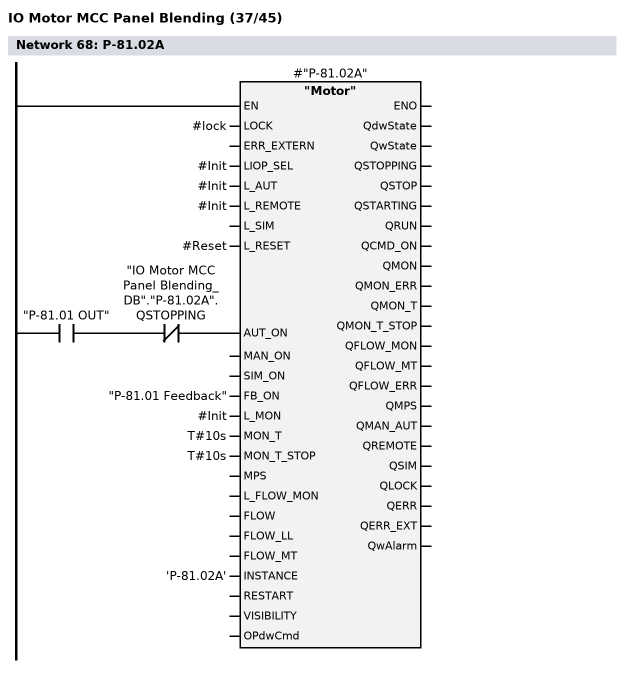
   RUNG wire#powerrail
      #"P-81.02A"(AUT_ON := wire#w1, LOCK := #lock, ERR_EXTERN :=, LIOP_SEL := #Init, L_AUT := #Init, L_REMOTE := #Init, L_SIM :=, L_RESET := #Reset, MAN_ON :=, SIM_ON :=, FB_ON := "P-81.01 Feedback", L_MON := #Init, MON_T := T#10s, MON_T_STOP := T#10s, MPS :=, L_FLOW_MON :=, FLOW :=, FLOW_LL :=, FLOW_MT :=, INSTANCE := 'P-81.02A', RESTART :=, VISIBILITY :=, OPdwCmd :=, QdwState =>, QwState =>, QSTOPPING =>, QSTOP =>, QSTARTING =>, QRUN =>, QCMD_ON =>, QMON =>, QMON_ERR =>, QMON_T =>, QMON_T_STOP =>, QFLOW_MON =>, QFLOW_MT =>, QFLOW_ERR =>, QMPS =>, QMAN_AUT =>, QREMOTE =>, QSIM =>, QLOCK =>, QERR =>, QERR_EXT =>, QwAlarm =>)
   END_RUNG
   RUNG wire#powerrail
      Contact( "P-81.01 OUT" )
      I_Contact( "IO Motor MCC Panel Blending_DB"."P-81.02A".QSTOPPING )
   END_RUNG wire#w1
   // the same network as SCL:
   #"P-81.02A"(LOCK := #lock,   // "Motor"
               LIOP_SEL := #Init,
               L_AUT := #Init,
               L_REMOTE := #Init,
               L_RESET := #Reset,
               AUT_ON := "P-81.01 OUT" AND NOT "IO Motor MCC Panel Blending_DB"."P-81.02A".QSTOPPING,
               FB_ON := "P-81.01 Feedback",
               L_MON := #Init,
               MON_T := T#10s,
               MON_T_STOP := T#10s,
               INSTANCE := 'P-81.02A');
END_REGION

REGION Network 69: P-81.02
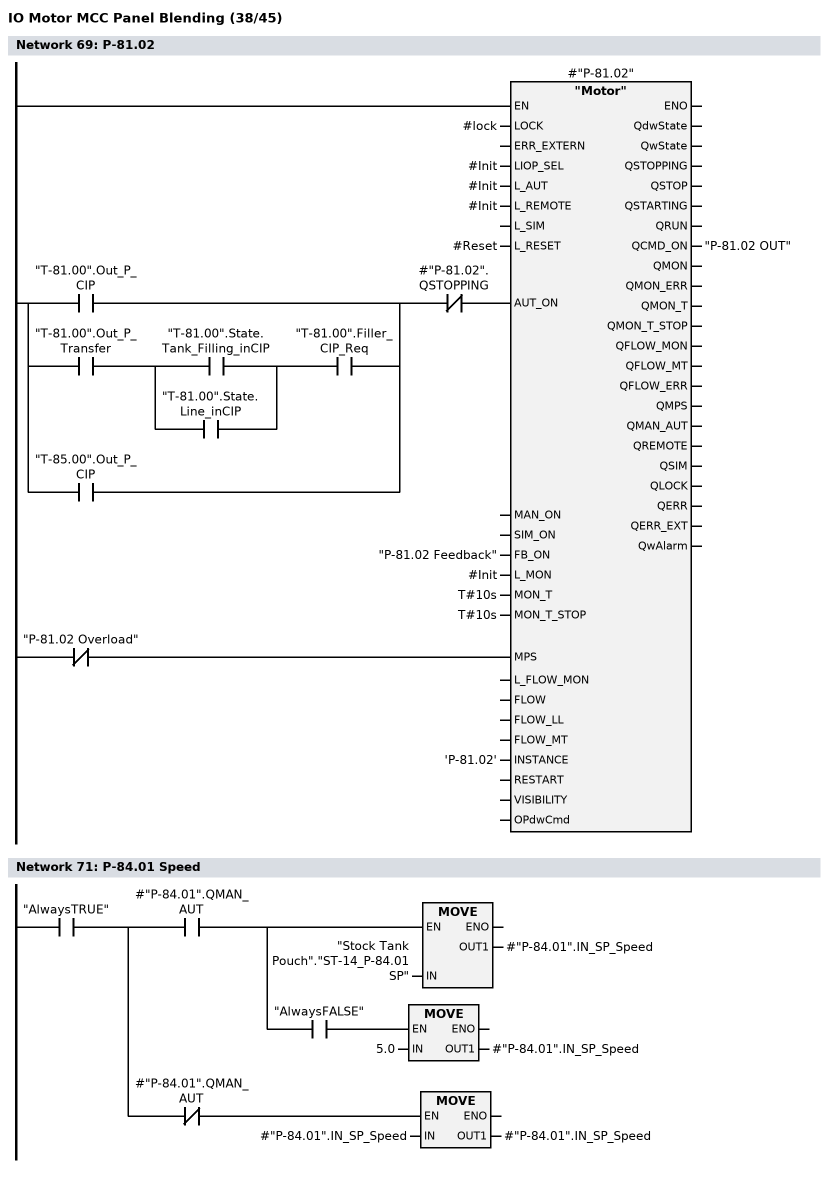
   RUNG wire#powerrail
      #"P-81.02"(AUT_ON := wire#w4, MPS := wire#w5, LOCK := #lock, ERR_EXTERN :=, LIOP_SEL := #Init, L_AUT := #Init, L_REMOTE := #Init, L_SIM :=, L_RESET := #Reset, MAN_ON :=, SIM_ON :=, FB_ON := "P-81.02 Feedback", L_MON := #Init, MON_T := T#10s, MON_T_STOP := T#10s, L_FLOW_MON :=, FLOW :=, FLOW_LL :=, FLOW_MT :=, INSTANCE := 'P-81.02', RESTART :=, VISIBILITY :=, OPdwCmd :=, QdwState =>, QwState =>, QSTOPPING =>, QSTOP =>, QSTARTING =>, QRUN =>, QCMD_ON => "P-81.02 OUT", QMON =>, QMON_ERR =>, QMON_T =>, QMON_T_STOP =>, QFLOW_MON =>, QFLOW_MT =>, QFLOW_ERR =>, QMPS =>, QMAN_AUT =>, QREMOTE =>, QSIM =>, QLOCK =>, QERR =>, QERR_EXT =>, QwAlarm =>)
   END_RUNG
   RUNG wire#powerrail
      Contact( "T-81.00".Out_P_CIP )
      wire#w1
      I_Contact( #"P-81.02".QSTOPPING )
   END_RUNG wire#w4
   RUNG wire#powerrail
      Contact( "T-81.00".Out_P_Transfer )
      wire#w2
      Contact( "T-81.00".State.Tank_Filling_inCIP )
      wire#w3
      Contact( "T-81.00".Filler_CIP_Req )
   END_RUNG wire#w1
   RUNG wire#w2
      Contact( "T-81.00".State.Line_inCIP )
   END_RUNG wire#w3
   RUNG wire#powerrail
      Contact( "T-85.00".Out_P_CIP )
   END_RUNG wire#w1
   RUNG wire#powerrail
      I_Contact( "P-81.02 Overload" )
   END_RUNG wire#w5
   // the same network as SCL:
   #"P-81.02"(LOCK := #lock,   // "Motor"
              LIOP_SEL := #Init,
              L_AUT := #Init,
              L_REMOTE := #Init,
              L_RESET := #Reset,
              AUT_ON := ("T-81.00".Out_P_CIP OR ("T-81.00".Out_P_Transfer AND ("T-81.00".State.Tank_Filling_inCIP OR "T-81.00".State.Line_inCIP) AND "T-81.00".Filler_CIP_Req) OR "T-85.00".Out_P_CIP) AND NOT #"P-81.02".QSTOPPING,
              FB_ON := "P-81.02 Feedback",
              L_MON := #Init,
              MON_T := T#10s,
              MON_T_STOP := T#10s,
              MPS := NOT "P-81.02 Overload",
              INSTANCE := 'P-81.02',
              QCMD_ON => "P-81.02 OUT");
END_REGION

REGION Network 71: P-84.01 Speed
   RUNG wire#powerrail
      Contact( "AlwaysTRUE" )
      wire#w1
      Contact( #"P-84.01".QMAN_AUT )
      wire#w2
      Move(in := "Stock Tank Pouch"."ST-14_P-84.01 SP", out1 => #"P-84.01".IN_SP_Speed)
   END_RUNG
   RUNG wire#w2
      Contact( "AlwaysFALSE" )
      Move(in := 5.0, out1 => #"P-84.01".IN_SP_Speed)
   END_RUNG
   RUNG wire#w1
      I_Contact( #"P-84.01".QMAN_AUT )
      Move(in := #"P-84.01".IN_SP_Speed, out1 => #"P-84.01".IN_SP_Speed)
   END_RUNG
   // the same network as SCL:
   #_w1 := "AlwaysTRUE" AND #"P-84.01".QMAN_AUT;
   IF #_w1 THEN #"P-84.01".IN_SP_Speed := "Stock Tank Pouch"."ST-14_P-84.01 SP"; END_IF;
   IF #_w1 AND "AlwaysFALSE" THEN #"P-84.01".IN_SP_Speed := 5.0; END_IF;
   IF "AlwaysTRUE" AND NOT #"P-84.01".QMAN_AUT THEN #"P-84.01".IN_SP_Speed := #"P-84.01".IN_SP_Speed; END_IF;
END_REGION

REGION Network 72: P-84.01
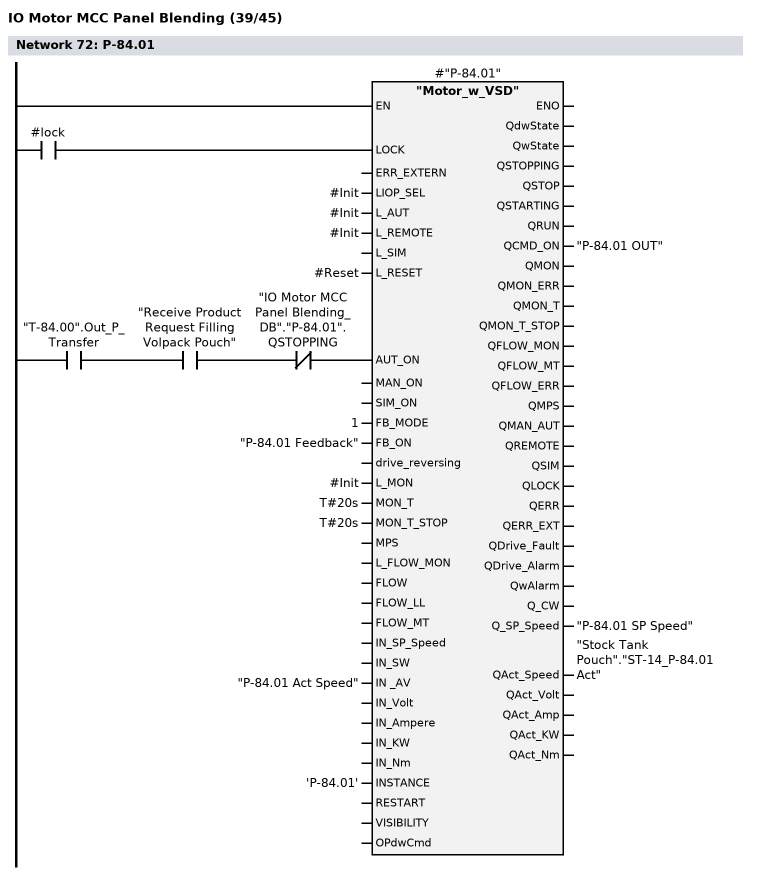
   RUNG wire#powerrail
      #"P-84.01"(LOCK := wire#w1, AUT_ON := wire#w2, ERR_EXTERN :=, LIOP_SEL := #Init, L_AUT := #Init, L_REMOTE := #Init, L_SIM :=, L_RESET := #Reset, MAN_ON :=, SIM_ON :=, FB_MODE := 1, FB_ON := "P-84.01 Feedback", drive_reversing :=, L_MON := #Init, MON_T := T#20s, MON_T_STOP := T#20s, MPS :=, L_FLOW_MON :=, FLOW :=, FLOW_LL :=, FLOW_MT :=, IN_SP_Speed :=, IN_SW :=, "IN _AV" := "P-84.01 Act Speed", IN_Volt :=, IN_Ampere :=, IN_KW :=, IN_Nm :=, INSTANCE := 'P-84.01', RESTART :=, VISIBILITY :=, OPdwCmd :=, QdwState =>, QwState =>, QSTOPPING =>, QSTOP =>, QSTARTING =>, QRUN =>, QCMD_ON => "P-84.01 OUT", QMON =>, QMON_ERR =>, QMON_T =>, QMON_T_STOP =>, QFLOW_MON =>, QFLOW_MT =>, QFLOW_ERR =>, QMPS =>, QMAN_AUT =>, QREMOTE =>, QSIM =>, QLOCK =>, QERR =>, QERR_EXT =>, QDrive_Fault =>, QDrive_Alarm =>, QwAlarm =>, Q_CW =>, Q_SP_Speed => "P-84.01 SP Speed", QAct_Speed => "Stock Tank Pouch"."ST-14_P-84.01 Act", QAct_Volt =>, QAct_Amp =>, QAct_KW =>, QAct_Nm =>)
   END_RUNG
   RUNG wire#powerrail
      Contact( #lock )
   END_RUNG wire#w1
   RUNG wire#powerrail
      Contact( "T-84.00".Out_P_Transfer )
      Contact( "Receive Product Request Filling Volpack Pouch" )
      I_Contact( "IO Motor MCC Panel Blending_DB"."P-84.01".QSTOPPING )
   END_RUNG wire#w2
   // the same network as SCL:
   #"P-84.01"(LOCK := #lock,   // "Motor_w_VSD"
              LIOP_SEL := #Init,
              L_AUT := #Init,
              L_REMOTE := #Init,
              L_RESET := #Reset,
              AUT_ON := "T-84.00".Out_P_Transfer AND "Receive Product Request Filling Volpack Pouch" AND NOT "IO Motor MCC Panel Blending_DB"."P-84.01".QSTOPPING,
              FB_MODE := 1,
              FB_ON := "P-84.01 Feedback",
              L_MON := #Init,
              MON_T := T#20s,
              MON_T_STOP := T#20s,
              "IN _AV" := "P-84.01 Act Speed",
              INSTANCE := 'P-84.01',
              QCMD_ON => "P-84.01 OUT",
              Q_SP_Speed => "P-84.01 SP Speed",
              QAct_Speed => "Stock Tank Pouch"."ST-14_P-84.01 Act");
END_REGION

REGION Network 73: P-84.01A
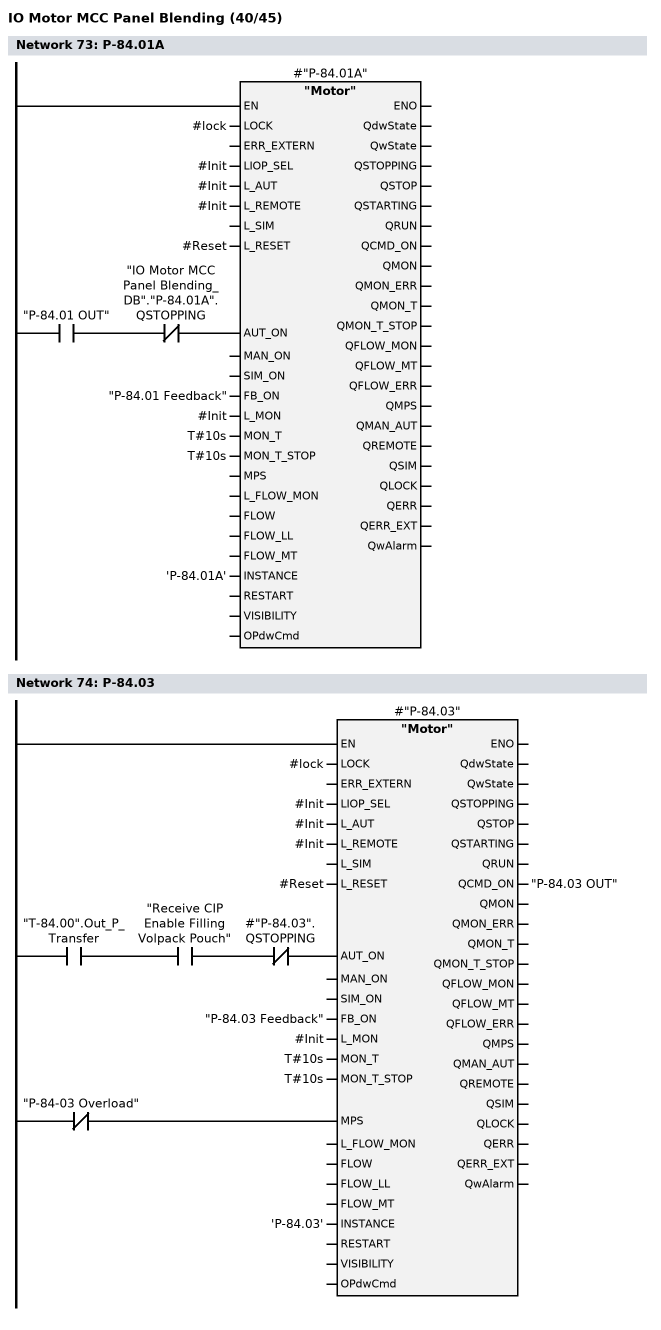
   RUNG wire#powerrail
      #"P-84.01A"(AUT_ON := wire#w1, LOCK := #lock, ERR_EXTERN :=, LIOP_SEL := #Init, L_AUT := #Init, L_REMOTE := #Init, L_SIM :=, L_RESET := #Reset, MAN_ON :=, SIM_ON :=, FB_ON := "P-84.01 Feedback", L_MON := #Init, MON_T := T#10s, MON_T_STOP := T#10s, MPS :=, L_FLOW_MON :=, FLOW :=, FLOW_LL :=, FLOW_MT :=, INSTANCE := 'P-84.01A', RESTART :=, VISIBILITY :=, OPdwCmd :=, QdwState =>, QwState =>, QSTOPPING =>, QSTOP =>, QSTARTING =>, QRUN =>, QCMD_ON =>, QMON =>, QMON_ERR =>, QMON_T =>, QMON_T_STOP =>, QFLOW_MON =>, QFLOW_MT =>, QFLOW_ERR =>, QMPS =>, QMAN_AUT =>, QREMOTE =>, QSIM =>, QLOCK =>, QERR =>, QERR_EXT =>, QwAlarm =>)
   END_RUNG
   RUNG wire#powerrail
      Contact( "P-84.01 OUT" )
      I_Contact( "IO Motor MCC Panel Blending_DB"."P-84.01A".QSTOPPING )
   END_RUNG wire#w1
   // the same network as SCL:
   #"P-84.01A"(LOCK := #lock,   // "Motor"
               LIOP_SEL := #Init,
               L_AUT := #Init,
               L_REMOTE := #Init,
               L_RESET := #Reset,
               AUT_ON := "P-84.01 OUT" AND NOT "IO Motor MCC Panel Blending_DB"."P-84.01A".QSTOPPING,
               FB_ON := "P-84.01 Feedback",
               L_MON := #Init,
               MON_T := T#10s,
               MON_T_STOP := T#10s,
               INSTANCE := 'P-84.01A');
END_REGION

REGION Network 74: P-84.03
   RUNG wire#powerrail
      #"P-84.03"(AUT_ON := wire#w1, MPS := wire#w2, LOCK := #lock, ERR_EXTERN :=, LIOP_SEL := #Init, L_AUT := #Init, L_REMOTE := #Init, L_SIM :=, L_RESET := #Reset, MAN_ON :=, SIM_ON :=, FB_ON := "P-84.03 Feedback", L_MON := #Init, MON_T := T#10s, MON_T_STOP := T#10s, L_FLOW_MON :=, FLOW :=, FLOW_LL :=, FLOW_MT :=, INSTANCE := 'P-84.03', RESTART :=, VISIBILITY :=, OPdwCmd :=, QdwState =>, QwState =>, QSTOPPING =>, QSTOP =>, QSTARTING =>, QRUN =>, QCMD_ON => "P-84.03 OUT", QMON =>, QMON_ERR =>, QMON_T =>, QMON_T_STOP =>, QFLOW_MON =>, QFLOW_MT =>, QFLOW_ERR =>, QMPS =>, QMAN_AUT =>, QREMOTE =>, QSIM =>, QLOCK =>, QERR =>, QERR_EXT =>, QwAlarm =>)
   END_RUNG
   RUNG wire#powerrail
      Contact( "T-84.00".Out_P_Transfer )
      Contact( "Receive CIP Enable Filling Volpack Pouch" )
      I_Contact( #"P-84.03".QSTOPPING )
   END_RUNG wire#w1
   RUNG wire#powerrail
      I_Contact( "P-84-03 Overload" )
   END_RUNG wire#w2
   // the same network as SCL:
   #"P-84.03"(LOCK := #lock,   // "Motor"
              LIOP_SEL := #Init,
              L_AUT := #Init,
              L_REMOTE := #Init,
              L_RESET := #Reset,
              AUT_ON := "T-84.00".Out_P_Transfer AND "Receive CIP Enable Filling Volpack Pouch" AND NOT #"P-84.03".QSTOPPING,
              FB_ON := "P-84.03 Feedback",
              L_MON := #Init,
              MON_T := T#10s,
              MON_T_STOP := T#10s,
              MPS := NOT "P-84-03 Overload",
              INSTANCE := 'P-84.03',
              QCMD_ON => "P-84.03 OUT");
END_REGION

REGION Network 75: P-84.02 Speed
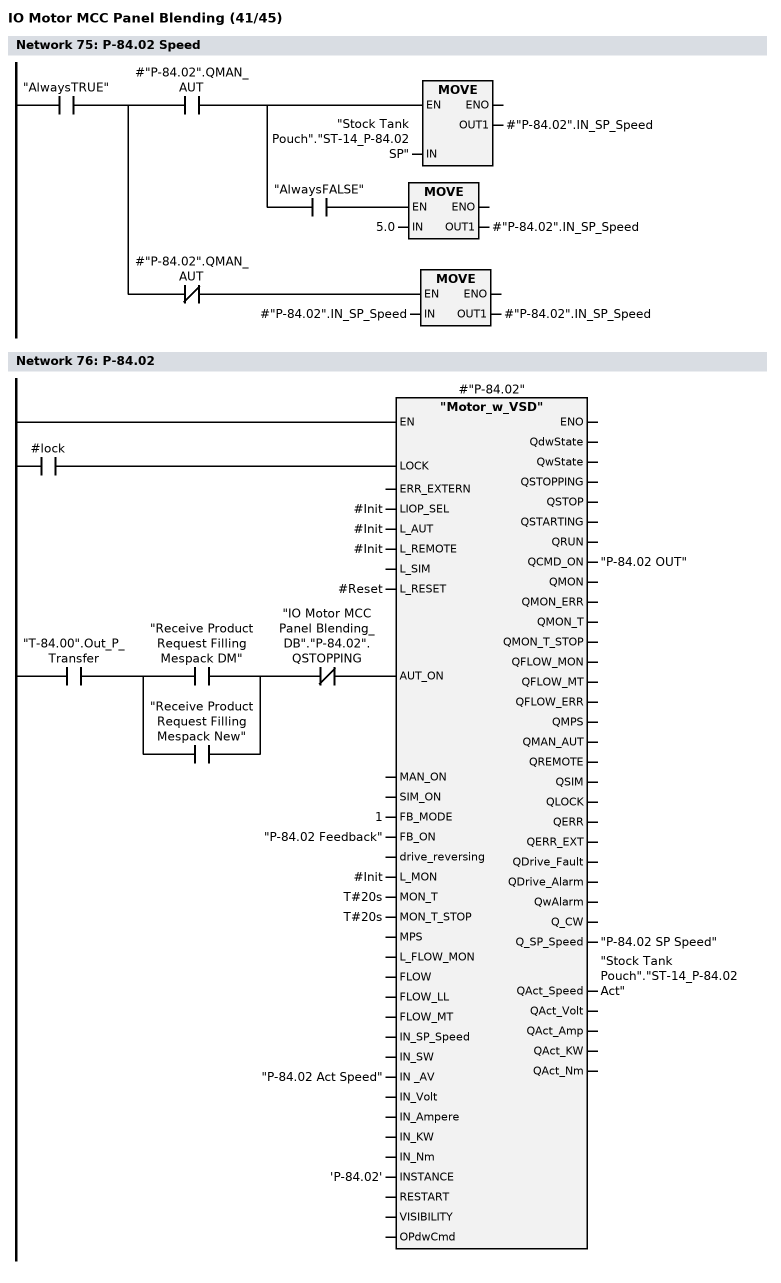
   RUNG wire#powerrail
      Contact( "AlwaysTRUE" )
      wire#w1
      Contact( #"P-84.02".QMAN_AUT )
      wire#w2
      Move(in := "Stock Tank Pouch"."ST-14_P-84.02 SP", out1 => #"P-84.02".IN_SP_Speed)
   END_RUNG
   RUNG wire#w2
      Contact( "AlwaysFALSE" )
      Move(in := 5.0, out1 => #"P-84.02".IN_SP_Speed)
   END_RUNG
   RUNG wire#w1
      I_Contact( #"P-84.02".QMAN_AUT )
      Move(in := #"P-84.02".IN_SP_Speed, out1 => #"P-84.02".IN_SP_Speed)
   END_RUNG
   // the same network as SCL:
   #_w1 := "AlwaysTRUE" AND #"P-84.02".QMAN_AUT;
   IF #_w1 THEN #"P-84.02".IN_SP_Speed := "Stock Tank Pouch"."ST-14_P-84.02 SP"; END_IF;
   IF #_w1 AND "AlwaysFALSE" THEN #"P-84.02".IN_SP_Speed := 5.0; END_IF;
   IF "AlwaysTRUE" AND NOT #"P-84.02".QMAN_AUT THEN #"P-84.02".IN_SP_Speed := #"P-84.02".IN_SP_Speed; END_IF;
END_REGION

REGION Network 76: P-84.02
   RUNG wire#powerrail
      #"P-84.02"(LOCK := wire#w1, AUT_ON := wire#w4, ERR_EXTERN :=, LIOP_SEL := #Init, L_AUT := #Init, L_REMOTE := #Init, L_SIM :=, L_RESET := #Reset, MAN_ON :=, SIM_ON :=, FB_MODE := 1, FB_ON := "P-84.02 Feedback", drive_reversing :=, L_MON := #Init, MON_T := T#20s, MON_T_STOP := T#20s, MPS :=, L_FLOW_MON :=, FLOW :=, FLOW_LL :=, FLOW_MT :=, IN_SP_Speed :=, IN_SW :=, "IN _AV" := "P-84.02 Act Speed", IN_Volt :=, IN_Ampere :=, IN_KW :=, IN_Nm :=, INSTANCE := 'P-84.02', RESTART :=, VISIBILITY :=, OPdwCmd :=, QdwState =>, QwState =>, QSTOPPING =>, QSTOP =>, QSTARTING =>, QRUN =>, QCMD_ON => "P-84.02 OUT", QMON =>, QMON_ERR =>, QMON_T =>, QMON_T_STOP =>, QFLOW_MON =>, QFLOW_MT =>, QFLOW_ERR =>, QMPS =>, QMAN_AUT =>, QREMOTE =>, QSIM =>, QLOCK =>, QERR =>, QERR_EXT =>, QDrive_Fault =>, QDrive_Alarm =>, QwAlarm =>, Q_CW =>, Q_SP_Speed => "P-84.02 SP Speed", QAct_Speed => "Stock Tank Pouch"."ST-14_P-84.02 Act", QAct_Volt =>, QAct_Amp =>, QAct_KW =>, QAct_Nm =>)
   END_RUNG
   RUNG wire#powerrail
      Contact( #lock )
   END_RUNG wire#w1
   RUNG wire#powerrail
      Contact( "T-84.00".Out_P_Transfer )
      wire#w2
      Contact( "Receive Product Request Filling Mespack DM" )
      wire#w3
      I_Contact( "IO Motor MCC Panel Blending_DB"."P-84.02".QSTOPPING )
   END_RUNG wire#w4
   RUNG wire#w2
      Contact( "Receive Product Request Filling Mespack New" )
   END_RUNG wire#w3
   // the same network as SCL:
   #"P-84.02"(LOCK := #lock,   // "Motor_w_VSD"
              LIOP_SEL := #Init,
              L_AUT := #Init,
              L_REMOTE := #Init,
              L_RESET := #Reset,
              AUT_ON := "T-84.00".Out_P_Transfer AND ("Receive Product Request Filling Mespack DM" OR "Receive Product Request Filling Mespack New") AND NOT "IO Motor MCC Panel Blending_DB"."P-84.02".QSTOPPING,
              FB_MODE := 1,
              FB_ON := "P-84.02 Feedback",
              L_MON := #Init,
              MON_T := T#20s,
              MON_T_STOP := T#20s,
              "IN _AV" := "P-84.02 Act Speed",
              INSTANCE := 'P-84.02',
              QCMD_ON => "P-84.02 OUT",
              Q_SP_Speed => "P-84.02 SP Speed",
              QAct_Speed => "Stock Tank Pouch"."ST-14_P-84.02 Act");
END_REGION

REGION Network 77: P-84.02A
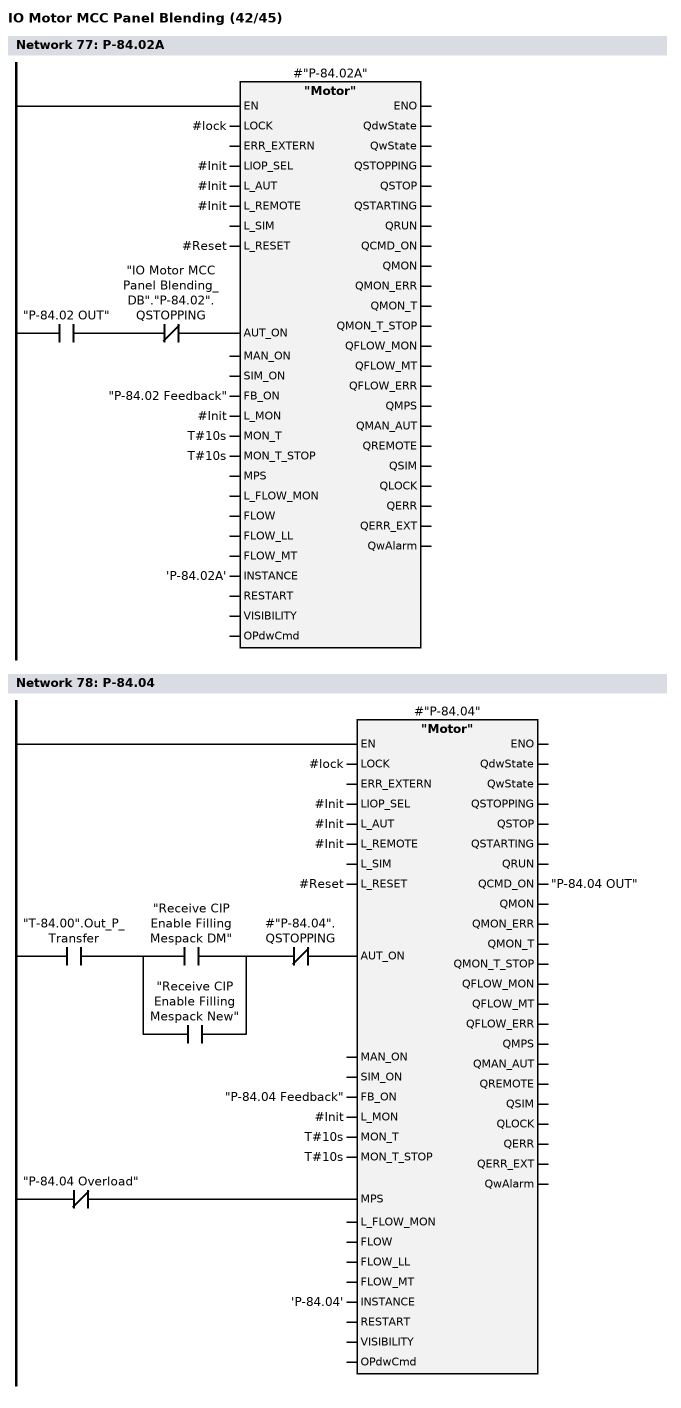
   RUNG wire#powerrail
      #"P-84.02A"(AUT_ON := wire#w1, LOCK := #lock, ERR_EXTERN :=, LIOP_SEL := #Init, L_AUT := #Init, L_REMOTE := #Init, L_SIM :=, L_RESET := #Reset, MAN_ON :=, SIM_ON :=, FB_ON := "P-84.02 Feedback", L_MON := #Init, MON_T := T#10s, MON_T_STOP := T#10s, MPS :=, L_FLOW_MON :=, FLOW :=, FLOW_LL :=, FLOW_MT :=, INSTANCE := 'P-84.02A', RESTART :=, VISIBILITY :=, OPdwCmd :=, QdwState =>, QwState =>, QSTOPPING =>, QSTOP =>, QSTARTING =>, QRUN =>, QCMD_ON =>, QMON =>, QMON_ERR =>, QMON_T =>, QMON_T_STOP =>, QFLOW_MON =>, QFLOW_MT =>, QFLOW_ERR =>, QMPS =>, QMAN_AUT =>, QREMOTE =>, QSIM =>, QLOCK =>, QERR =>, QERR_EXT =>, QwAlarm =>)
   END_RUNG
   RUNG wire#powerrail
      Contact( "P-84.02 OUT" )
      I_Contact( "IO Motor MCC Panel Blending_DB"."P-84.02".QSTOPPING )
   END_RUNG wire#w1
   // the same network as SCL:
   #"P-84.02A"(LOCK := #lock,   // "Motor"
               LIOP_SEL := #Init,
               L_AUT := #Init,
               L_REMOTE := #Init,
               L_RESET := #Reset,
               AUT_ON := "P-84.02 OUT" AND NOT "IO Motor MCC Panel Blending_DB"."P-84.02".QSTOPPING,
               FB_ON := "P-84.02 Feedback",
               L_MON := #Init,
               MON_T := T#10s,
               MON_T_STOP := T#10s,
               INSTANCE := 'P-84.02A');
END_REGION

REGION Network 78: P-84.04
   RUNG wire#powerrail
      #"P-84.04"(AUT_ON := wire#w3, MPS := wire#w4, LOCK := #lock, ERR_EXTERN :=, LIOP_SEL := #Init, L_AUT := #Init, L_REMOTE := #Init, L_SIM :=, L_RESET := #Reset, MAN_ON :=, SIM_ON :=, FB_ON := "P-84.04 Feedback", L_MON := #Init, MON_T := T#10s, MON_T_STOP := T#10s, L_FLOW_MON :=, FLOW :=, FLOW_LL :=, FLOW_MT :=, INSTANCE := 'P-84.04', RESTART :=, VISIBILITY :=, OPdwCmd :=, QdwState =>, QwState =>, QSTOPPING =>, QSTOP =>, QSTARTING =>, QRUN =>, QCMD_ON => "P-84.04 OUT", QMON =>, QMON_ERR =>, QMON_T =>, QMON_T_STOP =>, QFLOW_MON =>, QFLOW_MT =>, QFLOW_ERR =>, QMPS =>, QMAN_AUT =>, QREMOTE =>, QSIM =>, QLOCK =>, QERR =>, QERR_EXT =>, QwAlarm =>)
   END_RUNG
   RUNG wire#powerrail
      Contact( "T-84.00".Out_P_Transfer )
      wire#w1
      Contact( "Receive CIP Enable Filling Mespack DM" )
      wire#w2
      I_Contact( #"P-84.04".QSTOPPING )
   END_RUNG wire#w3
   RUNG wire#w1
      Contact( "Receive CIP Enable Filling Mespack New" )
   END_RUNG wire#w2
   RUNG wire#powerrail
      I_Contact( "P-84.04 Overload" )
   END_RUNG wire#w4
   // the same network as SCL:
   #"P-84.04"(LOCK := #lock,   // "Motor"
              LIOP_SEL := #Init,
              L_AUT := #Init,
              L_REMOTE := #Init,
              L_RESET := #Reset,
              AUT_ON := "T-84.00".Out_P_Transfer AND ("Receive CIP Enable Filling Mespack DM" OR "Receive CIP Enable Filling Mespack New") AND NOT #"P-84.04".QSTOPPING,
              FB_ON := "P-84.04 Feedback",
              L_MON := #Init,
              MON_T := T#10s,
              MON_T_STOP := T#10s,
              MPS := NOT "P-84.04 Overload",
              INSTANCE := 'P-84.04',
              QCMD_ON => "P-84.04 OUT");
END_REGION

REGION Network 80: P-82.01 Speed
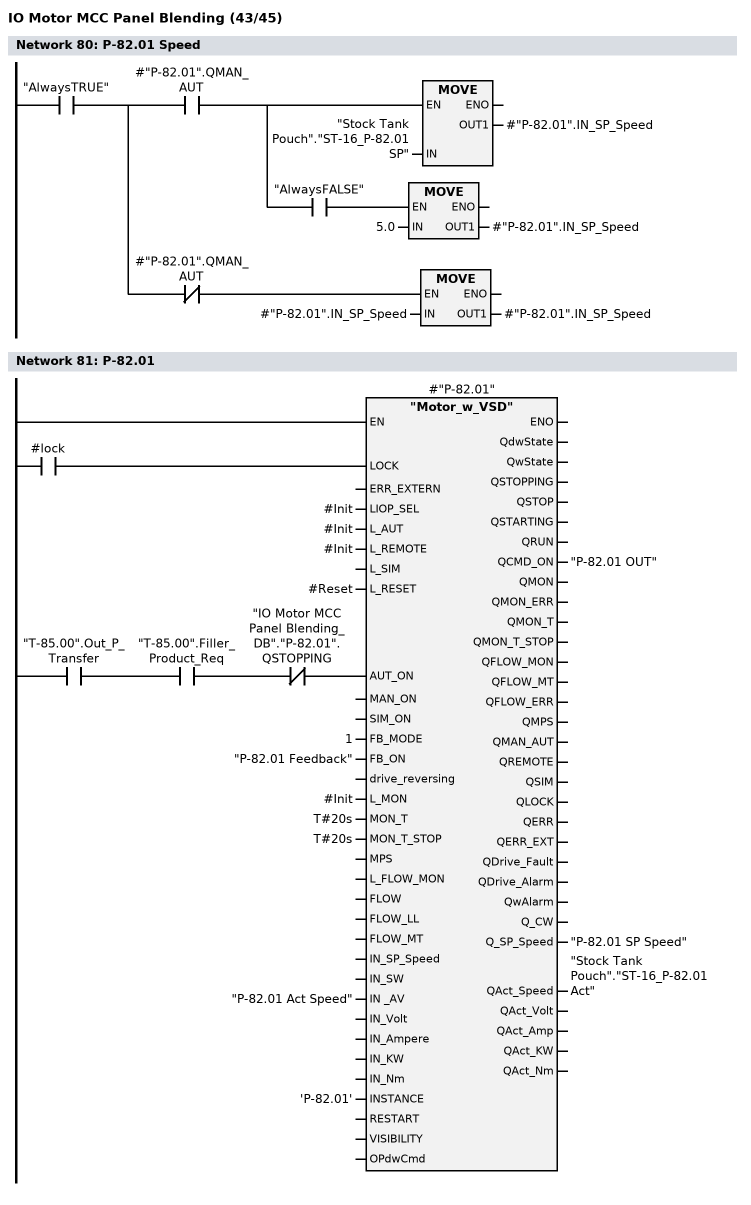
   RUNG wire#powerrail
      Contact( "AlwaysTRUE" )
      wire#w1
      Contact( #"P-82.01".QMAN_AUT )
      wire#w2
      Move(in := "Stock Tank Pouch"."ST-16_P-82.01 SP", out1 => #"P-82.01".IN_SP_Speed)
   END_RUNG
   RUNG wire#w2
      Contact( "AlwaysFALSE" )
      Move(in := 5.0, out1 => #"P-82.01".IN_SP_Speed)
   END_RUNG
   RUNG wire#w1
      I_Contact( #"P-82.01".QMAN_AUT )
      Move(in := #"P-82.01".IN_SP_Speed, out1 => #"P-82.01".IN_SP_Speed)
   END_RUNG
   // the same network as SCL:
   #_w1 := "AlwaysTRUE" AND #"P-82.01".QMAN_AUT;
   IF #_w1 THEN #"P-82.01".IN_SP_Speed := "Stock Tank Pouch"."ST-16_P-82.01 SP"; END_IF;
   IF #_w1 AND "AlwaysFALSE" THEN #"P-82.01".IN_SP_Speed := 5.0; END_IF;
   IF "AlwaysTRUE" AND NOT #"P-82.01".QMAN_AUT THEN #"P-82.01".IN_SP_Speed := #"P-82.01".IN_SP_Speed; END_IF;
END_REGION

REGION Network 81: P-82.01
   RUNG wire#powerrail
      #"P-82.01"(LOCK := wire#w1, AUT_ON := wire#w2, ERR_EXTERN :=, LIOP_SEL := #Init, L_AUT := #Init, L_REMOTE := #Init, L_SIM :=, L_RESET := #Reset, MAN_ON :=, SIM_ON :=, FB_MODE := 1, FB_ON := "P-82.01 Feedback", drive_reversing :=, L_MON := #Init, MON_T := T#20s, MON_T_STOP := T#20s, MPS :=, L_FLOW_MON :=, FLOW :=, FLOW_LL :=, FLOW_MT :=, IN_SP_Speed :=, IN_SW :=, "IN _AV" := "P-82.01 Act Speed", IN_Volt :=, IN_Ampere :=, IN_KW :=, IN_Nm :=, INSTANCE := 'P-82.01', RESTART :=, VISIBILITY :=, OPdwCmd :=, QdwState =>, QwState =>, QSTOPPING =>, QSTOP =>, QSTARTING =>, QRUN =>, QCMD_ON => "P-82.01 OUT", QMON =>, QMON_ERR =>, QMON_T =>, QMON_T_STOP =>, QFLOW_MON =>, QFLOW_MT =>, QFLOW_ERR =>, QMPS =>, QMAN_AUT =>, QREMOTE =>, QSIM =>, QLOCK =>, QERR =>, QERR_EXT =>, QDrive_Fault =>, QDrive_Alarm =>, QwAlarm =>, Q_CW =>, Q_SP_Speed => "P-82.01 SP Speed", QAct_Speed => "Stock Tank Pouch"."ST-16_P-82.01 Act", QAct_Volt =>, QAct_Amp =>, QAct_KW =>, QAct_Nm =>)
   END_RUNG
   RUNG wire#powerrail
      Contact( #lock )
   END_RUNG wire#w1
   RUNG wire#powerrail
      Contact( "T-85.00".Out_P_Transfer )
      Contact( "T-85.00".Filler_Product_Req )
      I_Contact( "IO Motor MCC Panel Blending_DB"."P-82.01".QSTOPPING )
   END_RUNG wire#w2
   // the same network as SCL:
   #"P-82.01"(LOCK := #lock,   // "Motor_w_VSD"
              LIOP_SEL := #Init,
              L_AUT := #Init,
              L_REMOTE := #Init,
              L_RESET := #Reset,
              AUT_ON := "T-85.00".Out_P_Transfer AND "T-85.00".Filler_Product_Req AND NOT "IO Motor MCC Panel Blending_DB"."P-82.01".QSTOPPING,
              FB_MODE := 1,
              FB_ON := "P-82.01 Feedback",
              L_MON := #Init,
              MON_T := T#20s,
              MON_T_STOP := T#20s,
              "IN _AV" := "P-82.01 Act Speed",
              INSTANCE := 'P-82.01',
              QCMD_ON => "P-82.01 OUT",
              Q_SP_Speed => "P-82.01 SP Speed",
              QAct_Speed => "Stock Tank Pouch"."ST-16_P-82.01 Act");
END_REGION

REGION Network 82: P-82.01A
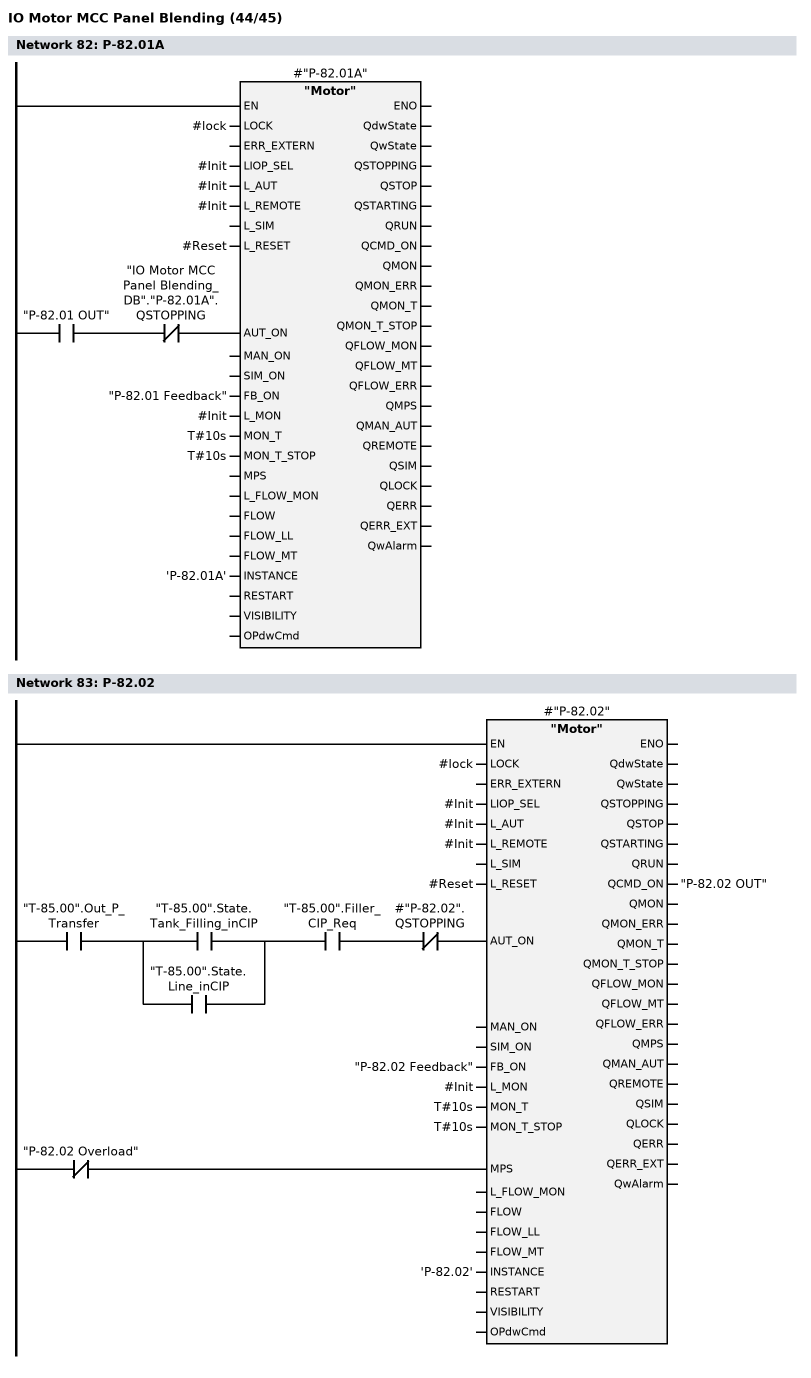
   RUNG wire#powerrail
      #"P-82.01A"(AUT_ON := wire#w1, LOCK := #lock, ERR_EXTERN :=, LIOP_SEL := #Init, L_AUT := #Init, L_REMOTE := #Init, L_SIM :=, L_RESET := #Reset, MAN_ON :=, SIM_ON :=, FB_ON := "P-82.01 Feedback", L_MON := #Init, MON_T := T#10s, MON_T_STOP := T#10s, MPS :=, L_FLOW_MON :=, FLOW :=, FLOW_LL :=, FLOW_MT :=, INSTANCE := 'P-82.01A', RESTART :=, VISIBILITY :=, OPdwCmd :=, QdwState =>, QwState =>, QSTOPPING =>, QSTOP =>, QSTARTING =>, QRUN =>, QCMD_ON =>, QMON =>, QMON_ERR =>, QMON_T =>, QMON_T_STOP =>, QFLOW_MON =>, QFLOW_MT =>, QFLOW_ERR =>, QMPS =>, QMAN_AUT =>, QREMOTE =>, QSIM =>, QLOCK =>, QERR =>, QERR_EXT =>, QwAlarm =>)
   END_RUNG
   RUNG wire#powerrail
      Contact( "P-82.01 OUT" )
      I_Contact( "IO Motor MCC Panel Blending_DB"."P-82.01A".QSTOPPING )
   END_RUNG wire#w1
   // the same network as SCL:
   #"P-82.01A"(LOCK := #lock,   // "Motor"
               LIOP_SEL := #Init,
               L_AUT := #Init,
               L_REMOTE := #Init,
               L_RESET := #Reset,
               AUT_ON := "P-82.01 OUT" AND NOT "IO Motor MCC Panel Blending_DB"."P-82.01A".QSTOPPING,
               FB_ON := "P-82.01 Feedback",
               L_MON := #Init,
               MON_T := T#10s,
               MON_T_STOP := T#10s,
               INSTANCE := 'P-82.01A');
END_REGION

REGION Network 83: P-82.02
   RUNG wire#powerrail
      #"P-82.02"(AUT_ON := wire#w3, MPS := wire#w4, LOCK := #lock, ERR_EXTERN :=, LIOP_SEL := #Init, L_AUT := #Init, L_REMOTE := #Init, L_SIM :=, L_RESET := #Reset, MAN_ON :=, SIM_ON :=, FB_ON := "P-82.02 Feedback", L_MON := #Init, MON_T := T#10s, MON_T_STOP := T#10s, L_FLOW_MON :=, FLOW :=, FLOW_LL :=, FLOW_MT :=, INSTANCE := 'P-82.02', RESTART :=, VISIBILITY :=, OPdwCmd :=, QdwState =>, QwState =>, QSTOPPING =>, QSTOP =>, QSTARTING =>, QRUN =>, QCMD_ON => "P-82.02 OUT", QMON =>, QMON_ERR =>, QMON_T =>, QMON_T_STOP =>, QFLOW_MON =>, QFLOW_MT =>, QFLOW_ERR =>, QMPS =>, QMAN_AUT =>, QREMOTE =>, QSIM =>, QLOCK =>, QERR =>, QERR_EXT =>, QwAlarm =>)
   END_RUNG
   RUNG wire#powerrail
      Contact( "T-85.00".Out_P_Transfer )
      wire#w1
      Contact( "T-85.00".State.Tank_Filling_inCIP )
      wire#w2
      Contact( "T-85.00".Filler_CIP_Req )
      I_Contact( #"P-82.02".QSTOPPING )
   END_RUNG wire#w3
   RUNG wire#w1
      Contact( "T-85.00".State.Line_inCIP )
   END_RUNG wire#w2
   RUNG wire#powerrail
      I_Contact( "P-82.02 Overload" )
   END_RUNG wire#w4
   // the same network as SCL:
   #"P-82.02"(LOCK := #lock,   // "Motor"
              LIOP_SEL := #Init,
              L_AUT := #Init,
              L_REMOTE := #Init,
              L_RESET := #Reset,
              AUT_ON := "T-85.00".Out_P_Transfer AND ("T-85.00".State.Tank_Filling_inCIP OR "T-85.00".State.Line_inCIP) AND "T-85.00".Filler_CIP_Req AND NOT #"P-82.02".QSTOPPING,
              FB_ON := "P-82.02 Feedback",
              L_MON := #Init,
              MON_T := T#10s,
              MON_T_STOP := T#10s,
              MPS := NOT "P-82.02 Overload",
              INSTANCE := 'P-82.02',
              QCMD_ON => "P-82.02 OUT");
END_REGION

REGION Network 84: XA-82.00
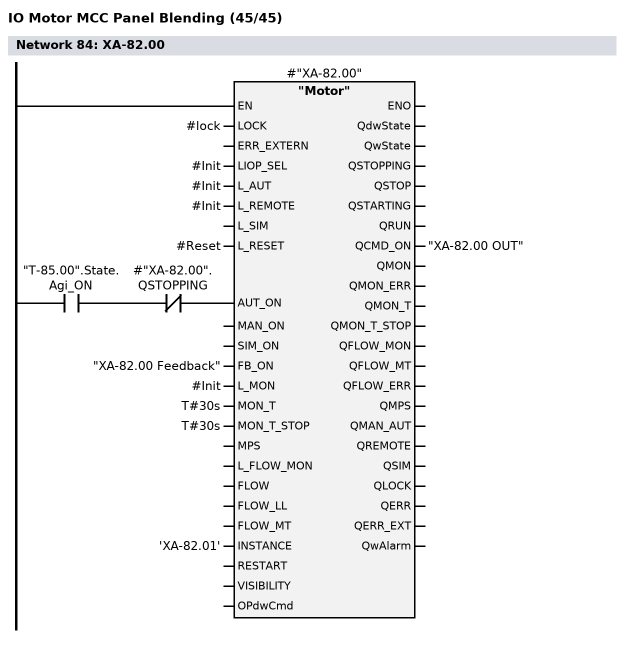
   RUNG wire#powerrail
      #"XA-82.00"(AUT_ON := wire#w1, LOCK := #lock, ERR_EXTERN :=, LIOP_SEL := #Init, L_AUT := #Init, L_REMOTE := #Init, L_SIM :=, L_RESET := #Reset, MAN_ON :=, SIM_ON :=, FB_ON := "XA-82.00 Feedback", L_MON := #Init, MON_T := T#30s, MON_T_STOP := T#30s, MPS :=, L_FLOW_MON :=, FLOW :=, FLOW_LL :=, FLOW_MT :=, INSTANCE := 'XA-82.01', RESTART :=, VISIBILITY :=, OPdwCmd :=, QdwState =>, QwState =>, QSTOPPING =>, QSTOP =>, QSTARTING =>, QRUN =>, QCMD_ON => "XA-82.00 OUT", QMON =>, QMON_ERR =>, QMON_T =>, QMON_T_STOP =>, QFLOW_MON =>, QFLOW_MT =>, QFLOW_ERR =>, QMPS =>, QMAN_AUT =>, QREMOTE =>, QSIM =>, QLOCK =>, QERR =>, QERR_EXT =>, QwAlarm =>)
   END_RUNG
   RUNG wire#powerrail
      Contact( "T-85.00".State.Agi_ON )
      I_Contact( #"XA-82.00".QSTOPPING )
   END_RUNG wire#w1
   // the same network as SCL:
   #"XA-82.00"(LOCK := #lock,   // "Motor"
               LIOP_SEL := #Init,
               L_AUT := #Init,
               L_REMOTE := #Init,
               L_RESET := #Reset,
               AUT_ON := "T-85.00".State.Agi_ON AND NOT #"XA-82.00".QSTOPPING,
               FB_ON := "XA-82.00 Feedback",
               L_MON := #Init,
               MON_T := T#30s,
               MON_T_STOP := T#30s,
               INSTANCE := 'XA-82.01',
               QCMD_ON => "XA-82.00 OUT");
END_REGION
END_FUNCTION_BLOCK

ORGANIZATION_BLOCK "Cyclic interrupt"   // OB30, LAD, CyclicInterrupt
{ S7_Optimized_Access := 'TRUE' }
VERSION : 0.1
// stored: AutoNumber true, IsIECCheckEnabled false, SetENOAutomatically false
   VAR_INPUT
      Initial_Call : Bool;   // Initial call of this OB
      Event_Count : Int;   // Events discarded
   END_VAR
   VAR_TEMP   // added for the SCL form of the ladder/FBD networks
      _w1 : Bool;
      _w2 : Bool;
      _w3 : Bool;
      _w4 : Bool;
      _w5 : Bool;
   END_VAR
BEGIN

REGION Network 1
   // "IO Analog Preparation_DB"."TT-01.01".QOUT
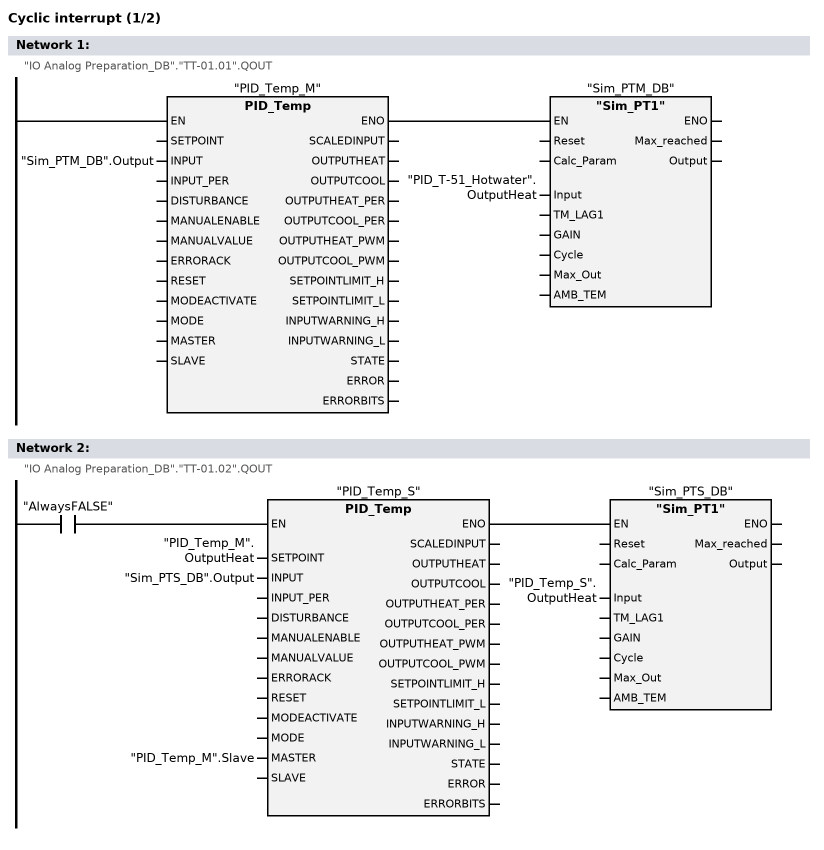
   RUNG wire#powerrail
      "PID_Temp_M".PID_Temp(Setpoint :=, Input := "Sim_PTM_DB".Output, Input_PER :=, Disturbance :=, ManualEnable :=, ManualValue :=, ErrorAck :=, Reset :=, ModeActivate :=, Mode :=, Master :=, Slave :=, ScaledInput =>, OutputHeat =>, OutputCool =>, OutputHeat_PER =>, OutputCool_PER =>, OutputHeat_PWM =>, OutputCool_PWM =>, SetpointLimit_H =>, SetpointLimit_L =>, InputWarning_H =>, InputWarning_L =>, State =>, Error =>, ErrorBits =>)
      "Sim_PTM_DB"(Reset :=, Calc_Param :=, Input := "PID_T-51_Hotwater".OutputHeat, TM_LAG1 :=, GAIN :=, Cycle :=, Max_Out :=, AMB_TEM :=, Max_reached =>, Output =>)
   END_RUNG
   // the same network as SCL:
   "PID_Temp_M"(Input := "Sim_PTM_DB".Output, ENO => #_w1);   // PID_Temp
   IF #_w1 THEN
       "Sim_PTM_DB"(Input := "PID_T-51_Hotwater".OutputHeat);   // "Sim_PT1"
   END_IF;
END_REGION

REGION Network 2
   // "IO Analog Preparation_DB"."TT-01.02".QOUT
   RUNG wire#powerrail
      Contact( "AlwaysFALSE" )
      "PID_Temp_S".PID_Temp(Setpoint := "PID_Temp_M".OutputHeat, Input := "Sim_PTS_DB".Output, Input_PER :=, Disturbance :=, ManualEnable :=, ManualValue :=, ErrorAck :=, Reset :=, ModeActivate :=, Mode :=, Master := "PID_Temp_M".Slave, Slave :=, ScaledInput =>, OutputHeat =>, OutputCool =>, OutputHeat_PER =>, OutputCool_PER =>, OutputHeat_PWM =>, OutputCool_PWM =>, SetpointLimit_H =>, SetpointLimit_L =>, InputWarning_H =>, InputWarning_L =>, State =>, Error =>, ErrorBits =>)
      "Sim_PTS_DB"(Reset :=, Calc_Param :=, Input := "PID_Temp_S".OutputHeat, TM_LAG1 :=, GAIN :=, Cycle :=, Max_Out :=, AMB_TEM :=, Max_reached =>, Output =>)
   END_RUNG
   // the same network as SCL:
   "PID_Temp_S"(EN := "AlwaysFALSE",   // PID_Temp
                Setpoint := "PID_Temp_M".OutputHeat,
                Input := "Sim_PTS_DB".Output,
                Master := "PID_Temp_M".Slave,
                ENO => #_w1);
   IF #_w1 THEN
       "Sim_PTS_DB"(Input := "PID_Temp_S".OutputHeat);   // "Sim_PT1"
   END_IF;
END_REGION

REGION Network 3: PID HotWater T51 Control
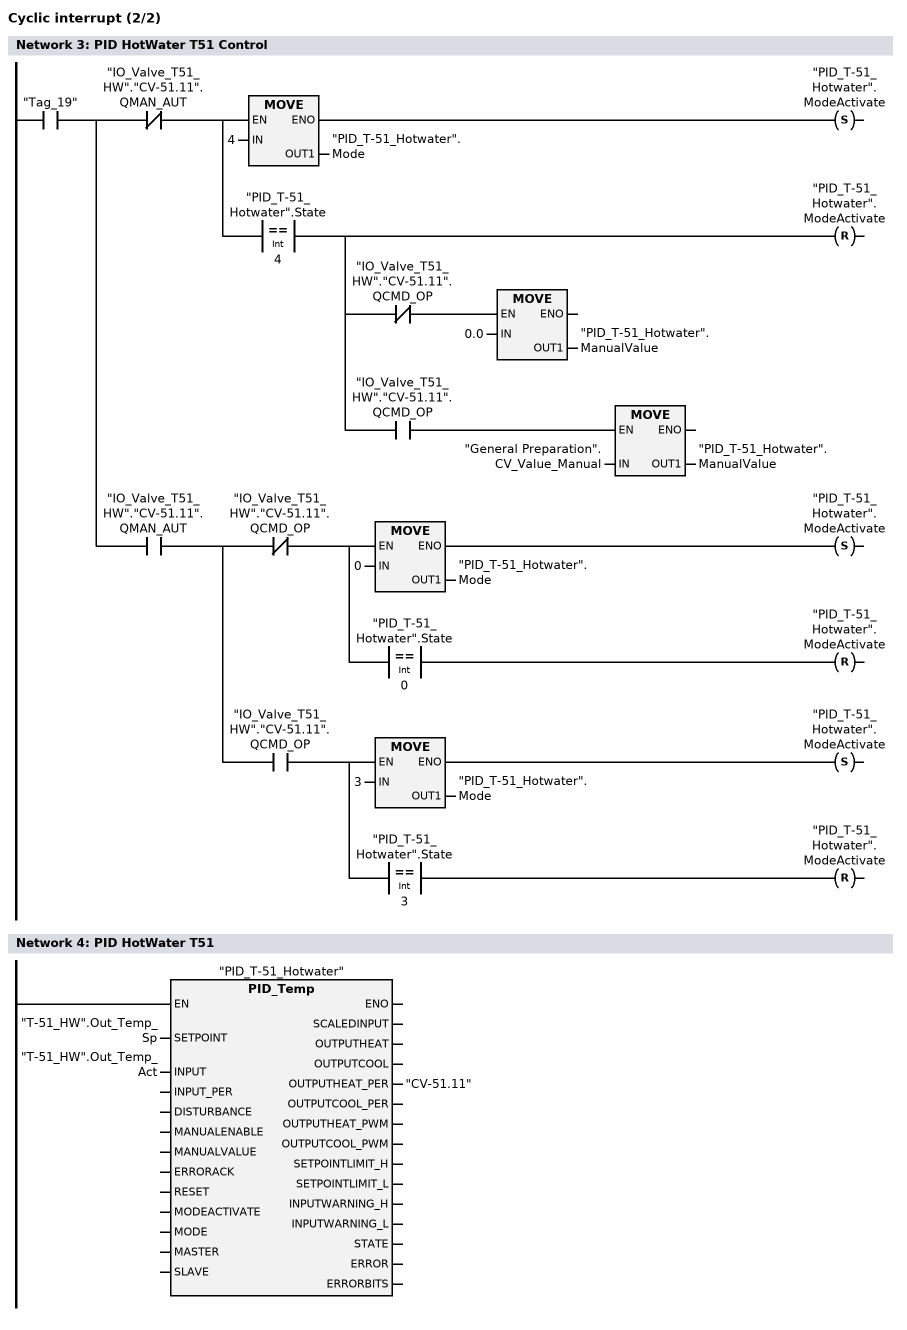
   RUNG wire#powerrail
      Contact( "Tag_19" )
      wire#w1
      I_Contact( "IO_Valve_T51_HW"."CV-51.11".QMAN_AUT )
      wire#w2
      Move(in := 4, out1 => "PID_T-51_Hotwater".Mode)
      S_Coil( "PID_T-51_Hotwater".ModeActivate )
   END_RUNG
   RUNG wire#w2
      { S7_Templates := "SrcType := Int" } EQ_Contact(in1 := "PID_T-51_Hotwater".State, in2 := 4)
      wire#w3
      R_Coil( "PID_T-51_Hotwater".ModeActivate )
   END_RUNG
   RUNG wire#w3
      I_Contact( "IO_Valve_T51_HW"."CV-51.11".QCMD_OP )
      Move(in := 0.0, out1 => "PID_T-51_Hotwater".ManualValue)
   END_RUNG
   RUNG wire#w3
      Contact( "IO_Valve_T51_HW"."CV-51.11".QCMD_OP )
      Move(in := "General Preparation".CV_Value_Manual, out1 => "PID_T-51_Hotwater".ManualValue)
   END_RUNG
   RUNG wire#w1
      Contact( "IO_Valve_T51_HW"."CV-51.11".QMAN_AUT )
      wire#w4
      I_Contact( "IO_Valve_T51_HW"."CV-51.11".QCMD_OP )
      wire#w5
      Move(in := 0, out1 => "PID_T-51_Hotwater".Mode)
      S_Coil( "PID_T-51_Hotwater".ModeActivate )
   END_RUNG
   RUNG wire#w5
      { S7_Templates := "SrcType := Int" } EQ_Contact(in1 := "PID_T-51_Hotwater".State, in2 := 0)
      R_Coil( "PID_T-51_Hotwater".ModeActivate )
   END_RUNG
   RUNG wire#w4
      Contact( "IO_Valve_T51_HW"."CV-51.11".QCMD_OP )
      wire#w6
      Move(in := 3, out1 => "PID_T-51_Hotwater".Mode)
      S_Coil( "PID_T-51_Hotwater".ModeActivate )
   END_RUNG
   RUNG wire#w6
      { S7_Templates := "SrcType := Int" } EQ_Contact(in1 := "PID_T-51_Hotwater".State, in2 := 3)
      R_Coil( "PID_T-51_Hotwater".ModeActivate )
   END_RUNG
   // the same network as SCL:
   #_w1 := "Tag_19" AND NOT "IO_Valve_T51_HW"."CV-51.11".QMAN_AUT;
   IF #_w1 THEN
       "PID_T-51_Hotwater".Mode := 4;
       "PID_T-51_Hotwater".ModeActivate := TRUE;
   END_IF;
   #_w2 := #_w1 AND ("PID_T-51_Hotwater".State = 4);
   IF #_w2 THEN "PID_T-51_Hotwater".ModeActivate := FALSE; END_IF;
   IF #_w2 AND NOT "IO_Valve_T51_HW"."CV-51.11".QCMD_OP THEN "PID_T-51_Hotwater".ManualValue := 0.0; END_IF;
   IF #_w2 AND "IO_Valve_T51_HW"."CV-51.11".QCMD_OP THEN
       "PID_T-51_Hotwater".ManualValue := "General Preparation".CV_Value_Manual;
   END_IF;
   #_w3 := "Tag_19" AND "IO_Valve_T51_HW"."CV-51.11".QMAN_AUT;
   #_w4 := #_w3 AND NOT "IO_Valve_T51_HW"."CV-51.11".QCMD_OP;
   IF #_w4 THEN
       "PID_T-51_Hotwater".Mode := 0;
       "PID_T-51_Hotwater".ModeActivate := TRUE;
   END_IF;
   IF #_w4 AND ("PID_T-51_Hotwater".State = 0) THEN "PID_T-51_Hotwater".ModeActivate := FALSE; END_IF;
   #_w5 := #_w3 AND "IO_Valve_T51_HW"."CV-51.11".QCMD_OP;
   IF #_w5 THEN
       "PID_T-51_Hotwater".Mode := 3;
       "PID_T-51_Hotwater".ModeActivate := TRUE;
   END_IF;
   IF #_w5 AND ("PID_T-51_Hotwater".State = 3) THEN "PID_T-51_Hotwater".ModeActivate := FALSE; END_IF;
END_REGION

REGION Network 4: PID HotWater T51
   RUNG wire#powerrail
      "PID_T-51_Hotwater".PID_Temp(Setpoint := "T-51_HW".Out_Temp_Sp, Input := "T-51_HW".Out_Temp_Act, Input_PER :=, Disturbance :=, ManualEnable :=, ManualValue :=, ErrorAck :=, Reset :=, ModeActivate :=, Mode :=, Master :=, Slave :=, ScaledInput =>, OutputHeat =>, OutputCool =>, OutputHeat_PER => "CV-51.11", OutputCool_PER =>, OutputHeat_PWM =>, OutputCool_PWM =>, SetpointLimit_H =>, SetpointLimit_L =>, InputWarning_H =>, InputWarning_L =>, State =>, Error =>, ErrorBits =>)
   END_RUNG
   // the same network as SCL:
   "PID_T-51_Hotwater"(Setpoint := "T-51_HW".Out_Temp_Sp,   // PID_Temp
                       Input := "T-51_HW".Out_Temp_Act,
                       OutputHeat_PER => "CV-51.11");
END_REGION
END_ORGANIZATION_BLOCK

FUNCTION_BLOCK "Sim_PT1"
{ S7_Optimized_Access := 'FALSE' }
VERSION : 0.1
   VAR_INPUT 
      Reset : Bool;
      Calc_Param : Bool;   // Übernimmt neue Parameter
      Input : Real;   // Input signal
      TM_LAG1 : Real := 1.0;   // Time Constant T1 [sek]
      GAIN : Real := 1.0;   // Proportionalitätskonstante
      Cycle : Real := 0.1;   // Tastzeit [sek]
      Max_Out : Real := 100.0;   // maximale Streckenbegrenzung
      AMB_TEM : Real;   // ambient temperature
   END_VAR

   VAR_OUTPUT 
      Max_reached : Bool;   // Strecke in der positiven Begrenzung
      Output : Real;   // Output signal
   END_VAR

   VAR 
      r_f1 : Real;
      r_e1 : Real;
      overfirst : Bool;
   END_VAR


BEGIN
	
	//**********************************************************************
	//  Simulation of a PT1-System
	//             GAIN
	//  F(p) = -----------
	//          TM_LAG*p + 1
	//  Call the simulation in a cyclic interrupt with
	//  T_Tast at least = T1/10!
	//**********************************************************************
	//
	IF #Calc_Param = True OR NOT #overfirst THEN
	  #overfirst := 1;
	  // Z-parameters For Laplace PT1-System
	  #r_e1 := - EXP(- #Cycle / #TM_LAG1);
	  #r_f1 := #GAIN * (1 + #r_e1);
	END_IF;
	
	// Differencial Equation of PT1-System
	//#Output := #Input*#r_f1 - #Output*#r_e1; // Original
	#Output := (#Input - #AMB_TEM) * #r_f1 - (#Output - #AMB_TEM) * #r_e1 + #AMB_TEM;
	
	// min limit of acutating variable and max-signal
	IF #Output > #Max_Out THEN
	  #Output := #Max_Out;
	  #Max_reached := True;
	ELSE
	  #Max_reached := False;
	END_IF;
	
	IF #Reset THEN
	  #Output := #AMB_TEM; //set output to AMB_TEM
	  //#Output := 0; // Original
	  
	END_IF;
	
	
	
END_FUNCTION_BLOCK

ORGANIZATION_BLOCK "IO access error"   // OB122, LAD, IOAccessError
{ S7_Optimized_Access := 'TRUE' }
VERSION : 0.1
// stored: IsIECCheckEnabled false, SetENOAutomatically false
   VAR_INPUT
      BlockNr : UInt;   // Number of causing block
      Reaction : USInt;   // 0:ignore, 1:substitute, 2:skip
      Fault_ID : Byte;   // 16#42:reading, 16#43:writing
      BlockType : USInt;   // 16#01:OB, 16#02:FC, 16#03:FB, 16#04:SFC, 16#05:SFB, 16#06:DB: Type of block causing the error
      Area : USInt;   // 16#81:I, 16#82:Q: IO area where the IOaccess error occured
      DBNr : DB_ANY;   // Reserved for system
      Csg_OBNr : OB_ANY;   // Number of OB causing the error
      Csg_Prio : USInt;   // Priority of OB causing the error
      Width : USInt;   // 0:bit, 1:byte, 2:word, 3:dword, 4:lword
   END_VAR
BEGIN
END_ORGANIZATION_BLOCK

ORGANIZATION_BLOCK "Programming error"   // OB121, LAD, ProgrammingError
{ S7_Optimized_Access := 'TRUE' }
VERSION : 0.1
// stored: IsIECCheckEnabled false, SetENOAutomatically false
   VAR_INPUT
      BlockNr : UInt;   // Number of causing block
      Reaction : USInt;   // 0:ignore, 1:substitute, 2:skip
      Fault_ID : Byte;   // Fault identifier
      BlockType : USInt;   // 16#01:OB, 16#02:FC, 16#03:FB, 16#04:SFC, 16#05:SFB, 16#06:DB: Type of block causing the error
      Area : USInt;   // Area where the error occured
      DBNr : DB_ANY;   // DB number if Area = DB or DI
      Csg_OBNr : OB_ANY;   // Number of OB causing the error
      Csg_Prio : USInt;   // Priority of OB causing the error
      Width : USInt;   // 0:bit, 1:byte, 2:word, 3:dword, 4:lword
   END_VAR
BEGIN
END_ORGANIZATION_BLOCK

ORGANIZATION_BLOCK "Rack or station failure"   // OB86, LAD, RackOrStationFailure
{ S7_Optimized_Access := 'TRUE' }
VERSION : 0.1
// stored: IsIECCheckEnabled false, SetENOAutomatically false
   VAR_INPUT
      LADDR : HW_DEVICE;   // Hardware identifier
      Event_Class : Byte;   // Event class
      Fault_ID : Byte;   // Fault identifier
   END_VAR
BEGIN
END_ORGANIZATION_BLOCK

ORGANIZATION_BLOCK "Startup"   // OB100, LAD, Startup
TITLE = "Complete Restart"
{ S7_Optimized_Access := 'TRUE' }
VERSION : 0.1
// stored: AutoNumber true, IsIECCheckEnabled false, SetENOAutomatically false
   VAR_INPUT
      LostRetentive : Bool;   // True if retentive data are lost
      LostRTC : Bool;   // True if date and time are lost
   END_VAR
BEGIN

REGION Network 1: initial
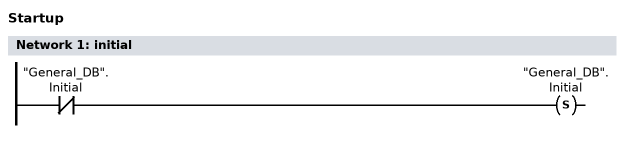
   RUNG wire#powerrail
      I_Contact( "General_DB".Initial )
      S_Coil( "General_DB".Initial )
   END_RUNG
   // the same network as SCL:
   IF NOT "General_DB".Initial THEN "General_DB".Initial := TRUE; END_IF;
END_REGION
END_ORGANIZATION_BLOCK

ORGANIZATION_BLOCK "Time error interrupt"   // OB80, LAD, TimeErrorInterrupt
{ S7_Optimized_Access := 'TRUE' }
VERSION : 0.1
// stored: IsIECCheckEnabled false, SetENOAutomatically false
   VAR_INPUT
      Fault_ID : Byte;   // Fault identifier
      Csg_OBnr : OB_ANY;   // Number of OB causing the error
      Csg_Prio : UInt;   // Priority of OB causing the error
   END_VAR
BEGIN
END_ORGANIZATION_BLOCK

ORGANIZATION_BLOCK "Totalizer_OB"   // OB31, LAD, CyclicInterrupt
{ S7_Optimized_Access := 'TRUE' }
VERSION : 0.1
// stored: AutoNumber false, IsIECCheckEnabled false, SetENOAutomatically false
   VAR_INPUT
      Initial_Call : Bool;   // Initial call of this OB
      Event_Count : Int;   // Events discarded
   END_VAR
   VAR_TEMP   // added for the SCL form of the ladder/FBD networks
      _w1 : Bool;
   END_VAR
BEGIN

REGION Network 1: Totalizer FT-00.01 Process Water Control
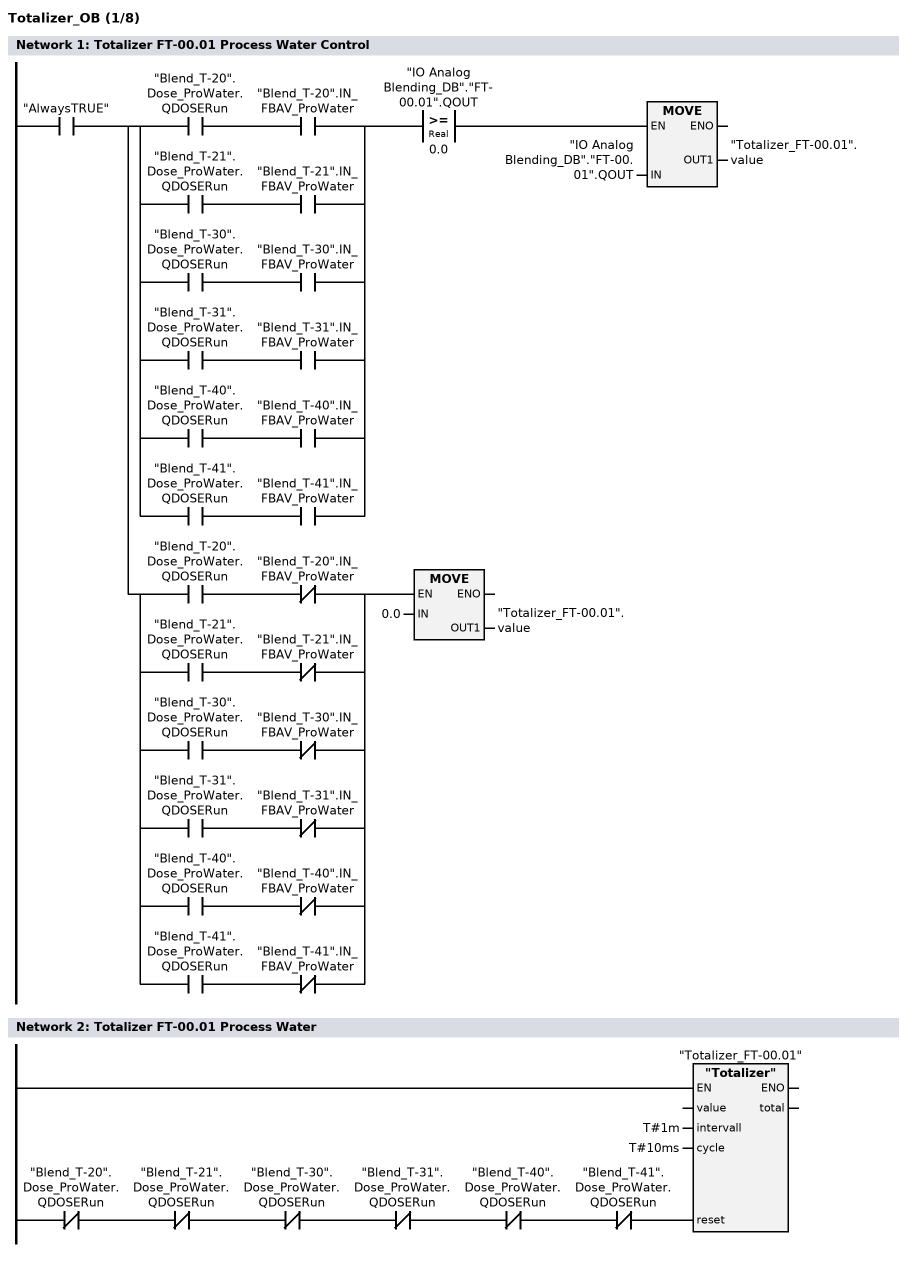
   RUNG wire#powerrail
      Contact( "AlwaysTRUE" )
      wire#w1
      Contact( "Blend_T-20".Dose_ProWater.QDOSERun )
      Contact( "Blend_T-20".IN_FBAV_ProWater )
      wire#w2
      { S7_Templates := "SrcType := Real" } GE_Contact(in1 := "IO Analog Blending_DB"."FT-00.01".QOUT, in2 := 0.0)
      Move(in := "IO Analog Blending_DB"."FT-00.01".QOUT, out1 => "Totalizer_FT-00.01".value)
   END_RUNG
   RUNG wire#w1
      Contact( "Blend_T-21".Dose_ProWater.QDOSERun )
      Contact( "Blend_T-21".IN_FBAV_ProWater )
   END_RUNG wire#w2
   RUNG wire#w1
      Contact( "Blend_T-30".Dose_ProWater.QDOSERun )
      Contact( "Blend_T-30".IN_FBAV_ProWater )
   END_RUNG wire#w2
   RUNG wire#w1
      Contact( "Blend_T-31".Dose_ProWater.QDOSERun )
      Contact( "Blend_T-31".IN_FBAV_ProWater )
   END_RUNG wire#w2
   RUNG wire#w1
      Contact( "Blend_T-40".Dose_ProWater.QDOSERun )
      Contact( "Blend_T-40".IN_FBAV_ProWater )
   END_RUNG wire#w2
   RUNG wire#w1
      Contact( "Blend_T-41".Dose_ProWater.QDOSERun )
      Contact( "Blend_T-41".IN_FBAV_ProWater )
   END_RUNG wire#w2
   RUNG wire#w1
      Contact( "Blend_T-20".Dose_ProWater.QDOSERun )
      I_Contact( "Blend_T-20".IN_FBAV_ProWater )
      wire#w3
      Move(in := 0.0, out1 => "Totalizer_FT-00.01".value)
   END_RUNG
   RUNG wire#w1
      Contact( "Blend_T-21".Dose_ProWater.QDOSERun )
      I_Contact( "Blend_T-21".IN_FBAV_ProWater )
   END_RUNG wire#w3
   RUNG wire#w1
      Contact( "Blend_T-30".Dose_ProWater.QDOSERun )
      I_Contact( "Blend_T-30".IN_FBAV_ProWater )
   END_RUNG wire#w3
   RUNG wire#w1
      Contact( "Blend_T-31".Dose_ProWater.QDOSERun )
      I_Contact( "Blend_T-31".IN_FBAV_ProWater )
   END_RUNG wire#w3
   RUNG wire#w1
      Contact( "Blend_T-40".Dose_ProWater.QDOSERun )
      I_Contact( "Blend_T-40".IN_FBAV_ProWater )
   END_RUNG wire#w3
   RUNG wire#w1
      Contact( "Blend_T-41".Dose_ProWater.QDOSERun )
      I_Contact( "Blend_T-41".IN_FBAV_ProWater )
   END_RUNG wire#w3
   // the same network as SCL:
   IF "AlwaysTRUE" AND (("Blend_T-20".Dose_ProWater.QDOSERun AND "Blend_T-20".IN_FBAV_ProWater) OR ("Blend_T-21".Dose_ProWater.QDOSERun AND "Blend_T-21".IN_FBAV_ProWater) OR ("Blend_T-30".Dose_ProWater.QDOSERun AND "Blend_T-30".IN_FBAV_ProWater) OR ("Blend_T-31".Dose_ProWater.QDOSERun AND "Blend_T-31".IN_FBAV_ProWater) OR ("Blend_T-40".Dose_ProWater.QDOSERun AND "Blend_T-40".IN_FBAV_ProWater) OR ("Blend_T-41".Dose_ProWater.QDOSERun AND "Blend_T-41".IN_FBAV_ProWater)) AND ("IO Analog Blending_DB"."FT-00.01".QOUT >= 0.0) THEN
       "Totalizer_FT-00.01".value := "IO Analog Blending_DB"."FT-00.01".QOUT;
   END_IF;
   IF "AlwaysTRUE" AND (("Blend_T-20".Dose_ProWater.QDOSERun AND NOT "Blend_T-20".IN_FBAV_ProWater) OR ("Blend_T-21".Dose_ProWater.QDOSERun AND NOT "Blend_T-21".IN_FBAV_ProWater) OR ("Blend_T-30".Dose_ProWater.QDOSERun AND NOT "Blend_T-30".IN_FBAV_ProWater) OR ("Blend_T-31".Dose_ProWater.QDOSERun AND NOT "Blend_T-31".IN_FBAV_ProWater) OR ("Blend_T-40".Dose_ProWater.QDOSERun AND NOT "Blend_T-40".IN_FBAV_ProWater) OR ("Blend_T-41".Dose_ProWater.QDOSERun AND NOT "Blend_T-41".IN_FBAV_ProWater)) THEN
       "Totalizer_FT-00.01".value := 0.0;
   END_IF;
END_REGION

REGION Network 2: Totalizer FT-00.01 Process Water
   RUNG wire#powerrail
      "Totalizer_FT-00.01"(reset := wire#w1, value :=, intervall := T#1m, cycle := T#10ms, total =>)
   END_RUNG
   RUNG wire#powerrail
      I_Contact( "Blend_T-20".Dose_ProWater.QDOSERun )
      I_Contact( "Blend_T-21".Dose_ProWater.QDOSERun )
      I_Contact( "Blend_T-30".Dose_ProWater.QDOSERun )
      I_Contact( "Blend_T-31".Dose_ProWater.QDOSERun )
      I_Contact( "Blend_T-40".Dose_ProWater.QDOSERun )
      I_Contact( "Blend_T-41".Dose_ProWater.QDOSERun )
   END_RUNG wire#w1
   // the same network as SCL:
   "Totalizer_FT-00.01"(intervall := T#1m,   // "Totalizer"
                        cycle := T#10ms,
                        reset := NOT "Blend_T-20".Dose_ProWater.QDOSERun AND NOT "Blend_T-21".Dose_ProWater.QDOSERun AND NOT "Blend_T-30".Dose_ProWater.QDOSERun AND NOT "Blend_T-31".Dose_ProWater.QDOSERun AND NOT "Blend_T-40".Dose_ProWater.QDOSERun AND NOT "Blend_T-41".Dose_ProWater.QDOSERun);
END_REGION

REGION Network 4: Totalizer FT.02.01 Chili Awetan 1 Control
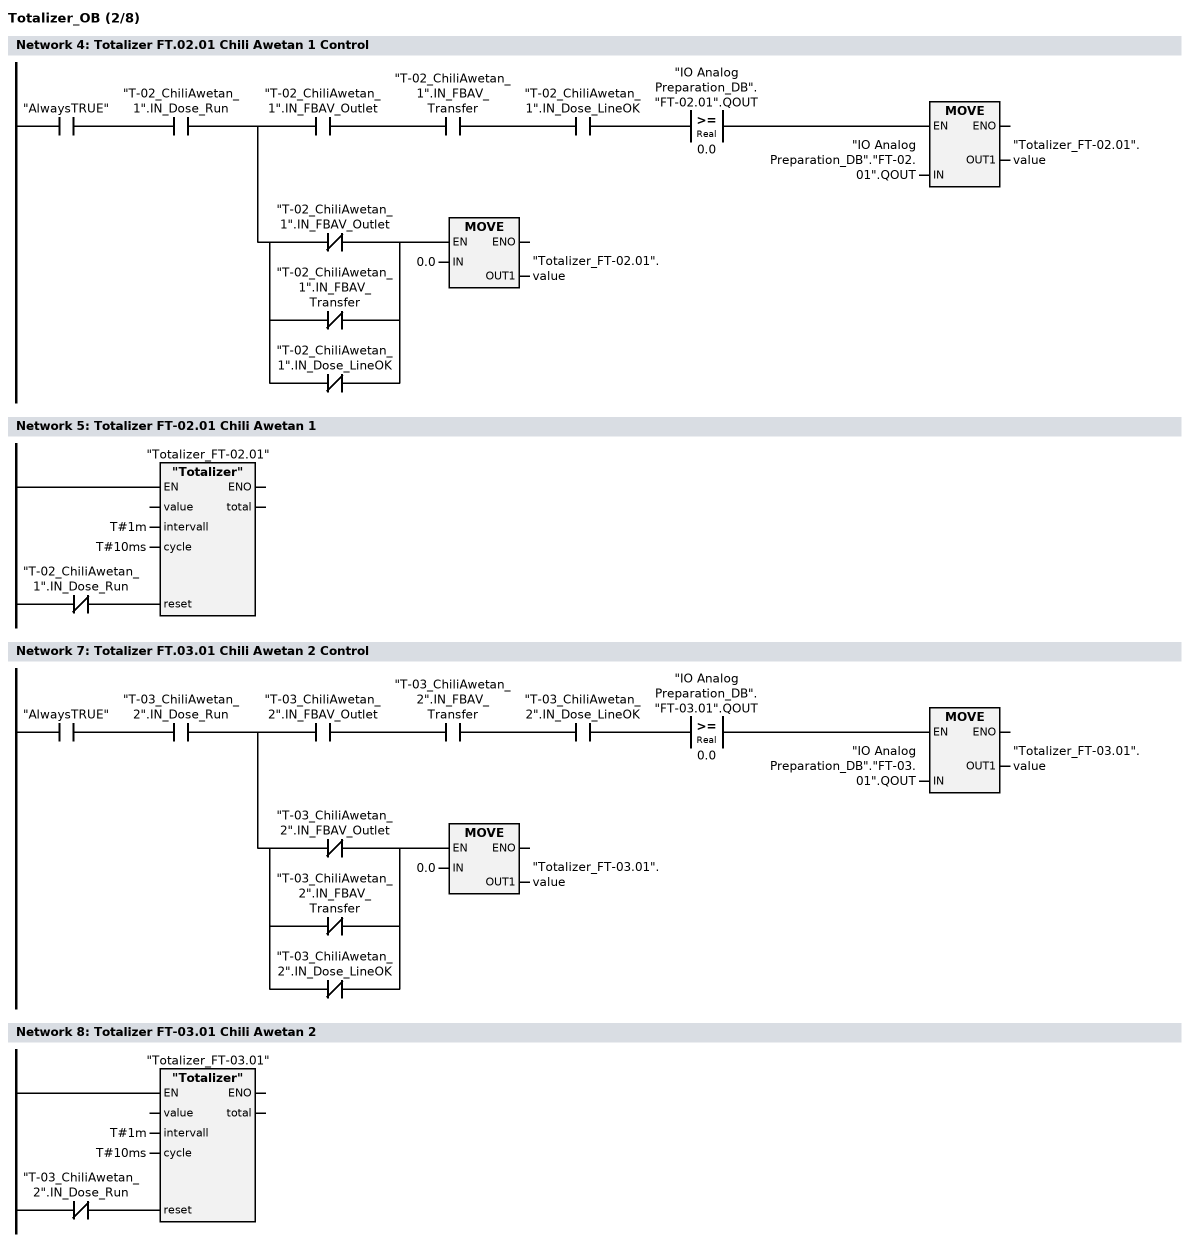
   RUNG wire#powerrail
      Contact( "AlwaysTRUE" )
      Contact( "T-02_ChiliAwetan_1".IN_Dose_Run )
      wire#w1
      Contact( "T-02_ChiliAwetan_1".IN_FBAV_Outlet )
      Contact( "T-02_ChiliAwetan_1".IN_FBAV_Transfer )
      Contact( "T-02_ChiliAwetan_1".IN_Dose_LineOK )
      { S7_Templates := "SrcType := Real" } GE_Contact(in1 := "IO Analog Preparation_DB"."FT-02.01".QOUT, in2 := 0.0)
      Move(in := "IO Analog Preparation_DB"."FT-02.01".QOUT, out1 => "Totalizer_FT-02.01".value)
   END_RUNG
   RUNG wire#w1
      I_Contact( "T-02_ChiliAwetan_1".IN_FBAV_Outlet )
      wire#w2
      Move(in := 0.0, out1 => "Totalizer_FT-02.01".value)
   END_RUNG
   RUNG wire#w1
      I_Contact( "T-02_ChiliAwetan_1".IN_FBAV_Transfer )
   END_RUNG wire#w2
   RUNG wire#w1
      I_Contact( "T-02_ChiliAwetan_1".IN_Dose_LineOK )
   END_RUNG wire#w2
   // the same network as SCL:
   #_w1 := "AlwaysTRUE" AND "T-02_ChiliAwetan_1".IN_Dose_Run;
   IF #_w1 AND "T-02_ChiliAwetan_1".IN_FBAV_Outlet AND "T-02_ChiliAwetan_1".IN_FBAV_Transfer AND "T-02_ChiliAwetan_1".IN_Dose_LineOK AND ("IO Analog Preparation_DB"."FT-02.01".QOUT >= 0.0) THEN
       "Totalizer_FT-02.01".value := "IO Analog Preparation_DB"."FT-02.01".QOUT;
   END_IF;
   IF #_w1 AND (NOT "T-02_ChiliAwetan_1".IN_FBAV_Outlet OR NOT "T-02_ChiliAwetan_1".IN_FBAV_Transfer OR NOT "T-02_ChiliAwetan_1".IN_Dose_LineOK) THEN
       "Totalizer_FT-02.01".value := 0.0;
   END_IF;
END_REGION

REGION Network 5: Totalizer FT-02.01 Chili Awetan 1
   RUNG wire#powerrail
      "Totalizer_FT-02.01"(reset := wire#w1, value :=, intervall := T#1m, cycle := T#10ms, total =>)
   END_RUNG
   RUNG wire#powerrail
      I_Contact( "T-02_ChiliAwetan_1".IN_Dose_Run )
   END_RUNG wire#w1
   // the same network as SCL:
   "Totalizer_FT-02.01"(intervall := T#1m, cycle := T#10ms, reset := NOT "T-02_ChiliAwetan_1".IN_Dose_Run);   // "Totalizer"
END_REGION

REGION Network 7: Totalizer FT.03.01 Chili Awetan 2 Control
   RUNG wire#powerrail
      Contact( "AlwaysTRUE" )
      Contact( "T-03_ChiliAwetan_2".IN_Dose_Run )
      wire#w1
      Contact( "T-03_ChiliAwetan_2".IN_FBAV_Outlet )
      Contact( "T-03_ChiliAwetan_2".IN_FBAV_Transfer )
      Contact( "T-03_ChiliAwetan_2".IN_Dose_LineOK )
      { S7_Templates := "SrcType := Real" } GE_Contact(in1 := "IO Analog Preparation_DB"."FT-03.01".QOUT, in2 := 0.0)
      Move(in := "IO Analog Preparation_DB"."FT-03.01".QOUT, out1 => "Totalizer_FT-03.01".value)
   END_RUNG
   RUNG wire#w1
      I_Contact( "T-03_ChiliAwetan_2".IN_FBAV_Outlet )
      wire#w2
      Move(in := 0.0, out1 => "Totalizer_FT-03.01".value)
   END_RUNG
   RUNG wire#w1
      I_Contact( "T-03_ChiliAwetan_2".IN_FBAV_Transfer )
   END_RUNG wire#w2
   RUNG wire#w1
      I_Contact( "T-03_ChiliAwetan_2".IN_Dose_LineOK )
   END_RUNG wire#w2
   // the same network as SCL:
   #_w1 := "AlwaysTRUE" AND "T-03_ChiliAwetan_2".IN_Dose_Run;
   IF #_w1 AND "T-03_ChiliAwetan_2".IN_FBAV_Outlet AND "T-03_ChiliAwetan_2".IN_FBAV_Transfer AND "T-03_ChiliAwetan_2".IN_Dose_LineOK AND ("IO Analog Preparation_DB"."FT-03.01".QOUT >= 0.0) THEN
       "Totalizer_FT-03.01".value := "IO Analog Preparation_DB"."FT-03.01".QOUT;
   END_IF;
   IF #_w1 AND (NOT "T-03_ChiliAwetan_2".IN_FBAV_Outlet OR NOT "T-03_ChiliAwetan_2".IN_FBAV_Transfer OR NOT "T-03_ChiliAwetan_2".IN_Dose_LineOK) THEN
       "Totalizer_FT-03.01".value := 0.0;
   END_IF;
END_REGION

REGION Network 8: Totalizer FT-03.01 Chili Awetan 2
   RUNG wire#powerrail
      "Totalizer_FT-03.01"(reset := wire#w1, value :=, intervall := T#1m, cycle := T#10ms, total =>)
   END_RUNG
   RUNG wire#powerrail
      I_Contact( "T-03_ChiliAwetan_2".IN_Dose_Run )
   END_RUNG wire#w1
   // the same network as SCL:
   "Totalizer_FT-03.01"(intervall := T#1m, cycle := T#10ms, reset := NOT "T-03_ChiliAwetan_2".IN_Dose_Run);   // "Totalizer"
END_REGION

REGION Network 10: Totalizer FT.04.01 Chili Awetan 3 Control
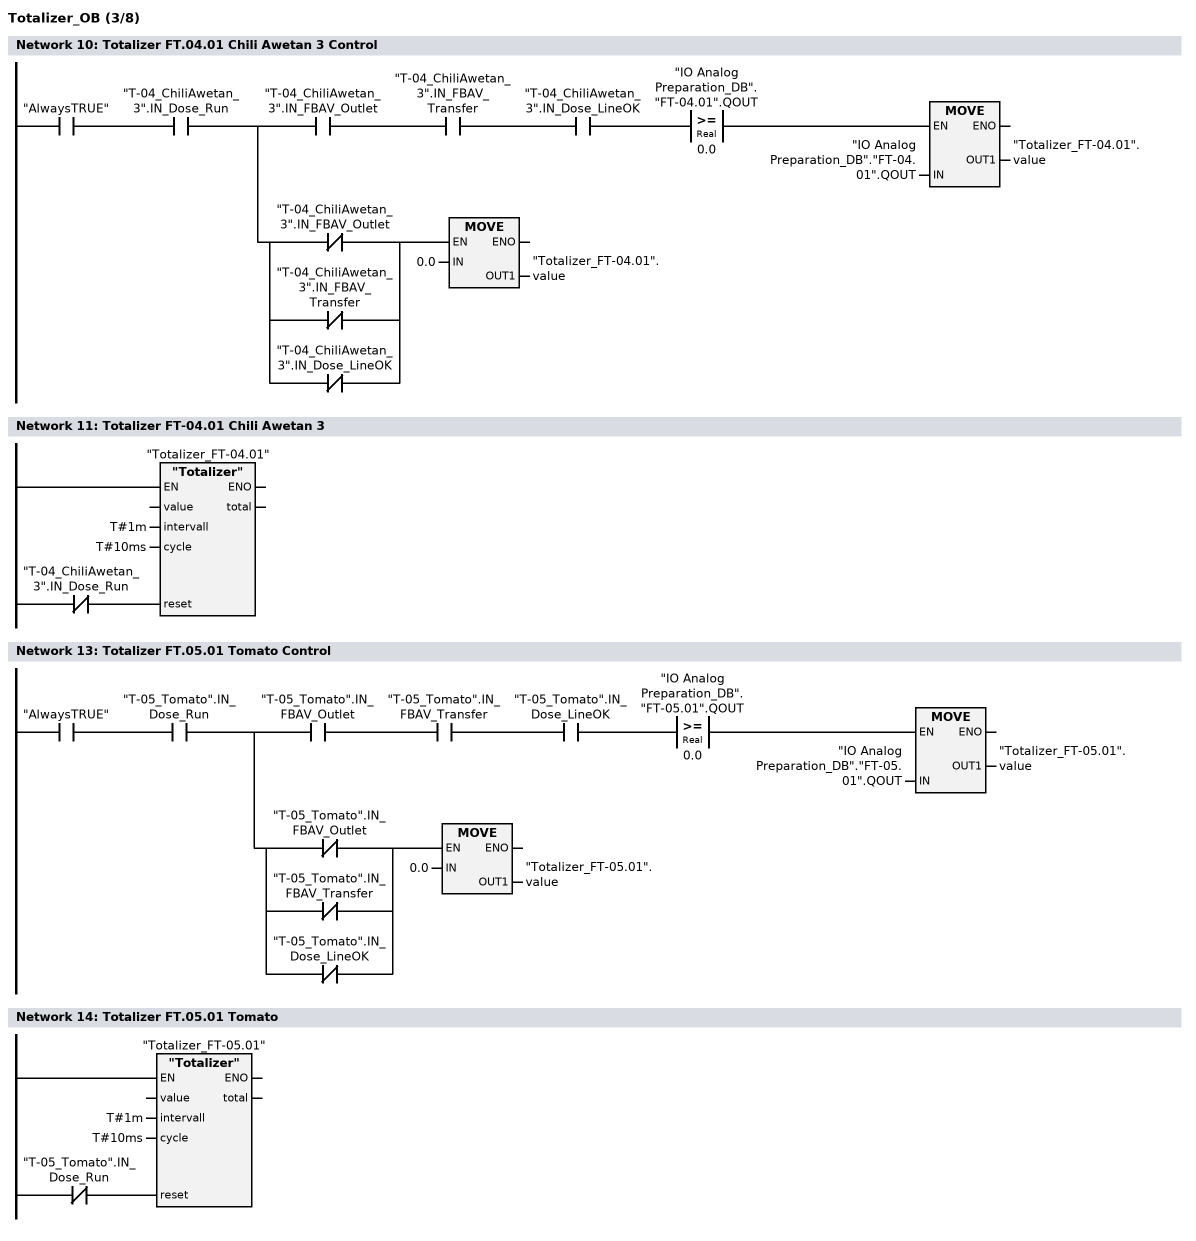
   RUNG wire#powerrail
      Contact( "AlwaysTRUE" )
      Contact( "T-04_ChiliAwetan_3".IN_Dose_Run )
      wire#w1
      Contact( "T-04_ChiliAwetan_3".IN_FBAV_Outlet )
      Contact( "T-04_ChiliAwetan_3".IN_FBAV_Transfer )
      Contact( "T-04_ChiliAwetan_3".IN_Dose_LineOK )
      { S7_Templates := "SrcType := Real" } GE_Contact(in1 := "IO Analog Preparation_DB"."FT-04.01".QOUT, in2 := 0.0)
      Move(in := "IO Analog Preparation_DB"."FT-04.01".QOUT, out1 => "Totalizer_FT-04.01".value)
   END_RUNG
   RUNG wire#w1
      I_Contact( "T-04_ChiliAwetan_3".IN_FBAV_Outlet )
      wire#w2
      Move(in := 0.0, out1 => "Totalizer_FT-04.01".value)
   END_RUNG
   RUNG wire#w1
      I_Contact( "T-04_ChiliAwetan_3".IN_FBAV_Transfer )
   END_RUNG wire#w2
   RUNG wire#w1
      I_Contact( "T-04_ChiliAwetan_3".IN_Dose_LineOK )
   END_RUNG wire#w2
   // the same network as SCL:
   #_w1 := "AlwaysTRUE" AND "T-04_ChiliAwetan_3".IN_Dose_Run;
   IF #_w1 AND "T-04_ChiliAwetan_3".IN_FBAV_Outlet AND "T-04_ChiliAwetan_3".IN_FBAV_Transfer AND "T-04_ChiliAwetan_3".IN_Dose_LineOK AND ("IO Analog Preparation_DB"."FT-04.01".QOUT >= 0.0) THEN
       "Totalizer_FT-04.01".value := "IO Analog Preparation_DB"."FT-04.01".QOUT;
   END_IF;
   IF #_w1 AND (NOT "T-04_ChiliAwetan_3".IN_FBAV_Outlet OR NOT "T-04_ChiliAwetan_3".IN_FBAV_Transfer OR NOT "T-04_ChiliAwetan_3".IN_Dose_LineOK) THEN
       "Totalizer_FT-04.01".value := 0.0;
   END_IF;
END_REGION

REGION Network 11: Totalizer FT-04.01 Chili Awetan 3
   RUNG wire#powerrail
      "Totalizer_FT-04.01"(reset := wire#w1, value :=, intervall := T#1m, cycle := T#10ms, total =>)
   END_RUNG
   RUNG wire#powerrail
      I_Contact( "T-04_ChiliAwetan_3".IN_Dose_Run )
   END_RUNG wire#w1
   // the same network as SCL:
   "Totalizer_FT-04.01"(intervall := T#1m, cycle := T#10ms, reset := NOT "T-04_ChiliAwetan_3".IN_Dose_Run);   // "Totalizer"
END_REGION

REGION Network 13: Totalizer FT.05.01 Tomato Control
   RUNG wire#powerrail
      Contact( "AlwaysTRUE" )
      Contact( "T-05_Tomato".IN_Dose_Run )
      wire#w1
      Contact( "T-05_Tomato".IN_FBAV_Outlet )
      Contact( "T-05_Tomato".IN_FBAV_Transfer )
      Contact( "T-05_Tomato".IN_Dose_LineOK )
      { S7_Templates := "SrcType := Real" } GE_Contact(in1 := "IO Analog Preparation_DB"."FT-05.01".QOUT, in2 := 0.0)
      Move(in := "IO Analog Preparation_DB"."FT-05.01".QOUT, out1 => "Totalizer_FT-05.01".value)
   END_RUNG
   RUNG wire#w1
      I_Contact( "T-05_Tomato".IN_FBAV_Outlet )
      wire#w2
      Move(in := 0.0, out1 => "Totalizer_FT-05.01".value)
   END_RUNG
   RUNG wire#w1
      I_Contact( "T-05_Tomato".IN_FBAV_Transfer )
   END_RUNG wire#w2
   RUNG wire#w1
      I_Contact( "T-05_Tomato".IN_Dose_LineOK )
   END_RUNG wire#w2
   // the same network as SCL:
   #_w1 := "AlwaysTRUE" AND "T-05_Tomato".IN_Dose_Run;
   IF #_w1 AND "T-05_Tomato".IN_FBAV_Outlet AND "T-05_Tomato".IN_FBAV_Transfer AND "T-05_Tomato".IN_Dose_LineOK AND ("IO Analog Preparation_DB"."FT-05.01".QOUT >= 0.0) THEN
       "Totalizer_FT-05.01".value := "IO Analog Preparation_DB"."FT-05.01".QOUT;
   END_IF;
   IF #_w1 AND (NOT "T-05_Tomato".IN_FBAV_Outlet OR NOT "T-05_Tomato".IN_FBAV_Transfer OR NOT "T-05_Tomato".IN_Dose_LineOK) THEN
       "Totalizer_FT-05.01".value := 0.0;
   END_IF;
END_REGION

REGION Network 14: Totalizer FT.05.01 Tomato
   RUNG wire#powerrail
      "Totalizer_FT-05.01"(reset := wire#w1, value :=, intervall := T#1m, cycle := T#10ms, total =>)
   END_RUNG
   RUNG wire#powerrail
      I_Contact( "T-05_Tomato".IN_Dose_Run )
   END_RUNG wire#w1
   // the same network as SCL:
   "Totalizer_FT-05.01"(intervall := T#1m, cycle := T#10ms, reset := NOT "T-05_Tomato".IN_Dose_Run);   // "Totalizer"
END_REGION

REGION Network 16: Totalizer FT.06.01 Chili Fresh 1 Control
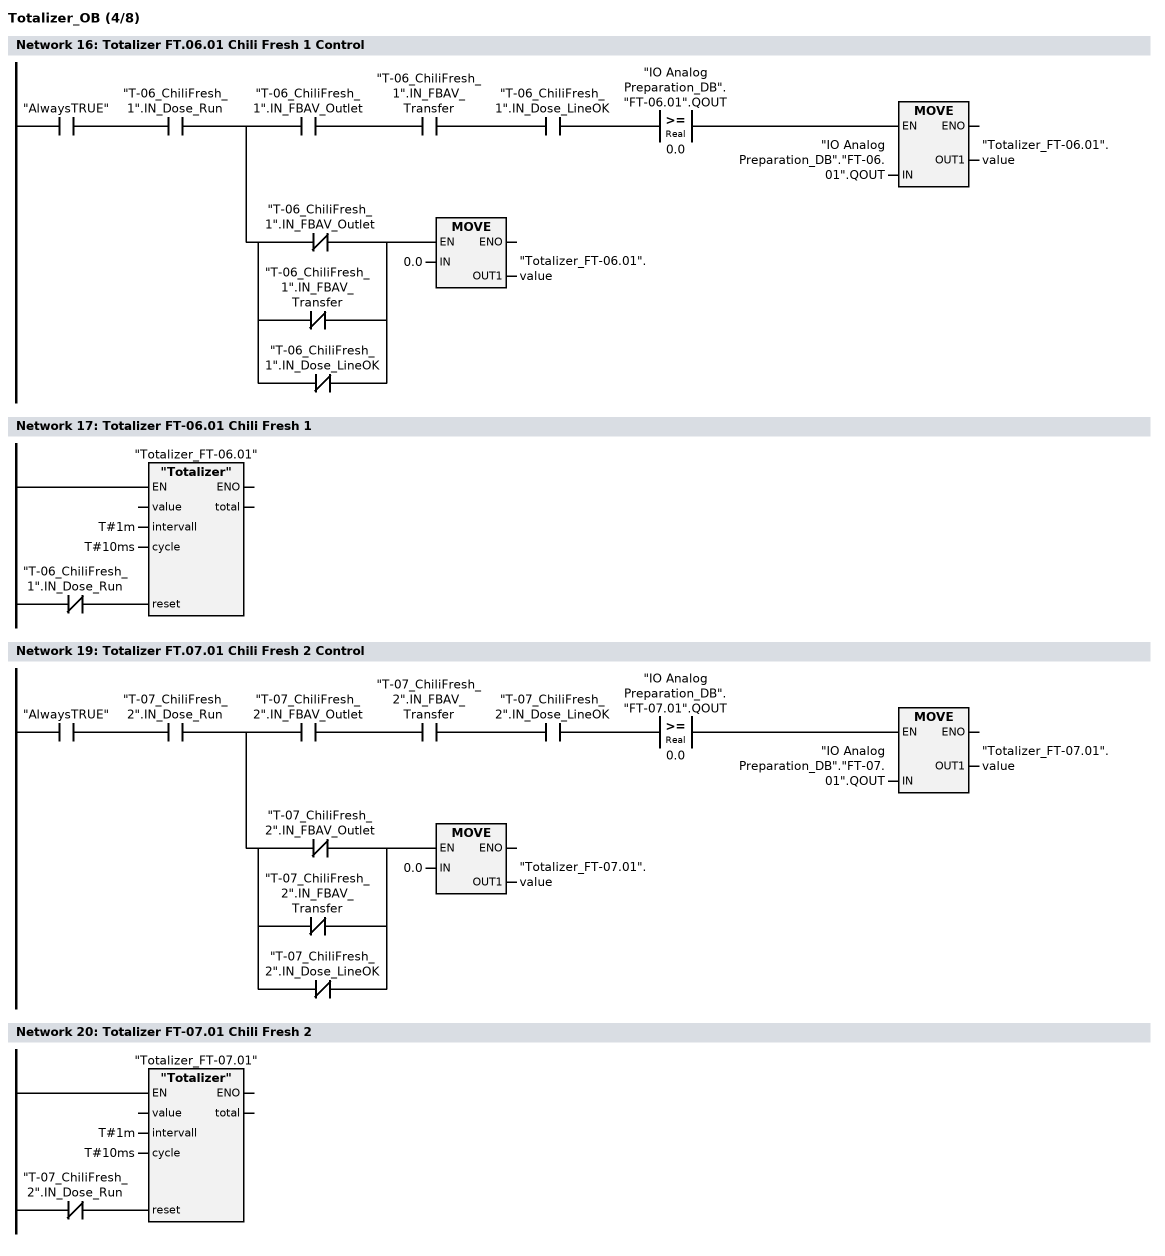
   RUNG wire#powerrail
      Contact( "AlwaysTRUE" )
      Contact( "T-06_ChiliFresh_1".IN_Dose_Run )
      wire#w1
      Contact( "T-06_ChiliFresh_1".IN_FBAV_Outlet )
      Contact( "T-06_ChiliFresh_1".IN_FBAV_Transfer )
      Contact( "T-06_ChiliFresh_1".IN_Dose_LineOK )
      { S7_Templates := "SrcType := Real" } GE_Contact(in1 := "IO Analog Preparation_DB"."FT-06.01".QOUT, in2 := 0.0)
      Move(in := "IO Analog Preparation_DB"."FT-06.01".QOUT, out1 => "Totalizer_FT-06.01".value)
   END_RUNG
   RUNG wire#w1
      I_Contact( "T-06_ChiliFresh_1".IN_FBAV_Outlet )
      wire#w2
      Move(in := 0.0, out1 => "Totalizer_FT-06.01".value)
   END_RUNG
   RUNG wire#w1
      I_Contact( "T-06_ChiliFresh_1".IN_FBAV_Transfer )
   END_RUNG wire#w2
   RUNG wire#w1
      I_Contact( "T-06_ChiliFresh_1".IN_Dose_LineOK )
   END_RUNG wire#w2
   // the same network as SCL:
   #_w1 := "AlwaysTRUE" AND "T-06_ChiliFresh_1".IN_Dose_Run;
   IF #_w1 AND "T-06_ChiliFresh_1".IN_FBAV_Outlet AND "T-06_ChiliFresh_1".IN_FBAV_Transfer AND "T-06_ChiliFresh_1".IN_Dose_LineOK AND ("IO Analog Preparation_DB"."FT-06.01".QOUT >= 0.0) THEN
       "Totalizer_FT-06.01".value := "IO Analog Preparation_DB"."FT-06.01".QOUT;
   END_IF;
   IF #_w1 AND (NOT "T-06_ChiliFresh_1".IN_FBAV_Outlet OR NOT "T-06_ChiliFresh_1".IN_FBAV_Transfer OR NOT "T-06_ChiliFresh_1".IN_Dose_LineOK) THEN
       "Totalizer_FT-06.01".value := 0.0;
   END_IF;
END_REGION

REGION Network 17: Totalizer FT-06.01 Chili Fresh 1
   RUNG wire#powerrail
      "Totalizer_FT-06.01"(reset := wire#w1, value :=, intervall := T#1m, cycle := T#10ms, total =>)
   END_RUNG
   RUNG wire#powerrail
      I_Contact( "T-06_ChiliFresh_1".IN_Dose_Run )
   END_RUNG wire#w1
   // the same network as SCL:
   "Totalizer_FT-06.01"(intervall := T#1m, cycle := T#10ms, reset := NOT "T-06_ChiliFresh_1".IN_Dose_Run);   // "Totalizer"
END_REGION

REGION Network 19: Totalizer FT.07.01 Chili Fresh 2 Control
   RUNG wire#powerrail
      Contact( "AlwaysTRUE" )
      Contact( "T-07_ChiliFresh_2".IN_Dose_Run )
      wire#w1
      Contact( "T-07_ChiliFresh_2".IN_FBAV_Outlet )
      Contact( "T-07_ChiliFresh_2".IN_FBAV_Transfer )
      Contact( "T-07_ChiliFresh_2".IN_Dose_LineOK )
      { S7_Templates := "SrcType := Real" } GE_Contact(in1 := "IO Analog Preparation_DB"."FT-07.01".QOUT, in2 := 0.0)
      Move(in := "IO Analog Preparation_DB"."FT-07.01".QOUT, out1 => "Totalizer_FT-07.01".value)
   END_RUNG
   RUNG wire#w1
      I_Contact( "T-07_ChiliFresh_2".IN_FBAV_Outlet )
      wire#w2
      Move(in := 0.0, out1 => "Totalizer_FT-07.01".value)
   END_RUNG
   RUNG wire#w1
      I_Contact( "T-07_ChiliFresh_2".IN_FBAV_Transfer )
   END_RUNG wire#w2
   RUNG wire#w1
      I_Contact( "T-07_ChiliFresh_2".IN_Dose_LineOK )
   END_RUNG wire#w2
   // the same network as SCL:
   #_w1 := "AlwaysTRUE" AND "T-07_ChiliFresh_2".IN_Dose_Run;
   IF #_w1 AND "T-07_ChiliFresh_2".IN_FBAV_Outlet AND "T-07_ChiliFresh_2".IN_FBAV_Transfer AND "T-07_ChiliFresh_2".IN_Dose_LineOK AND ("IO Analog Preparation_DB"."FT-07.01".QOUT >= 0.0) THEN
       "Totalizer_FT-07.01".value := "IO Analog Preparation_DB"."FT-07.01".QOUT;
   END_IF;
   IF #_w1 AND (NOT "T-07_ChiliFresh_2".IN_FBAV_Outlet OR NOT "T-07_ChiliFresh_2".IN_FBAV_Transfer OR NOT "T-07_ChiliFresh_2".IN_Dose_LineOK) THEN
       "Totalizer_FT-07.01".value := 0.0;
   END_IF;
END_REGION

REGION Network 20: Totalizer FT-07.01 Chili Fresh 2
   RUNG wire#powerrail
      "Totalizer_FT-07.01"(reset := wire#w1, value :=, intervall := T#1m, cycle := T#10ms, total =>)
   END_RUNG
   RUNG wire#powerrail
      I_Contact( "T-07_ChiliFresh_2".IN_Dose_Run )
   END_RUNG wire#w1
   // the same network as SCL:
   "Totalizer_FT-07.01"(intervall := T#1m, cycle := T#10ms, reset := NOT "T-07_ChiliFresh_2".IN_Dose_Run);   // "Totalizer"
END_REGION

REGION Network 22: Totalizer FT.08.01 Chili Fresh 3 Control
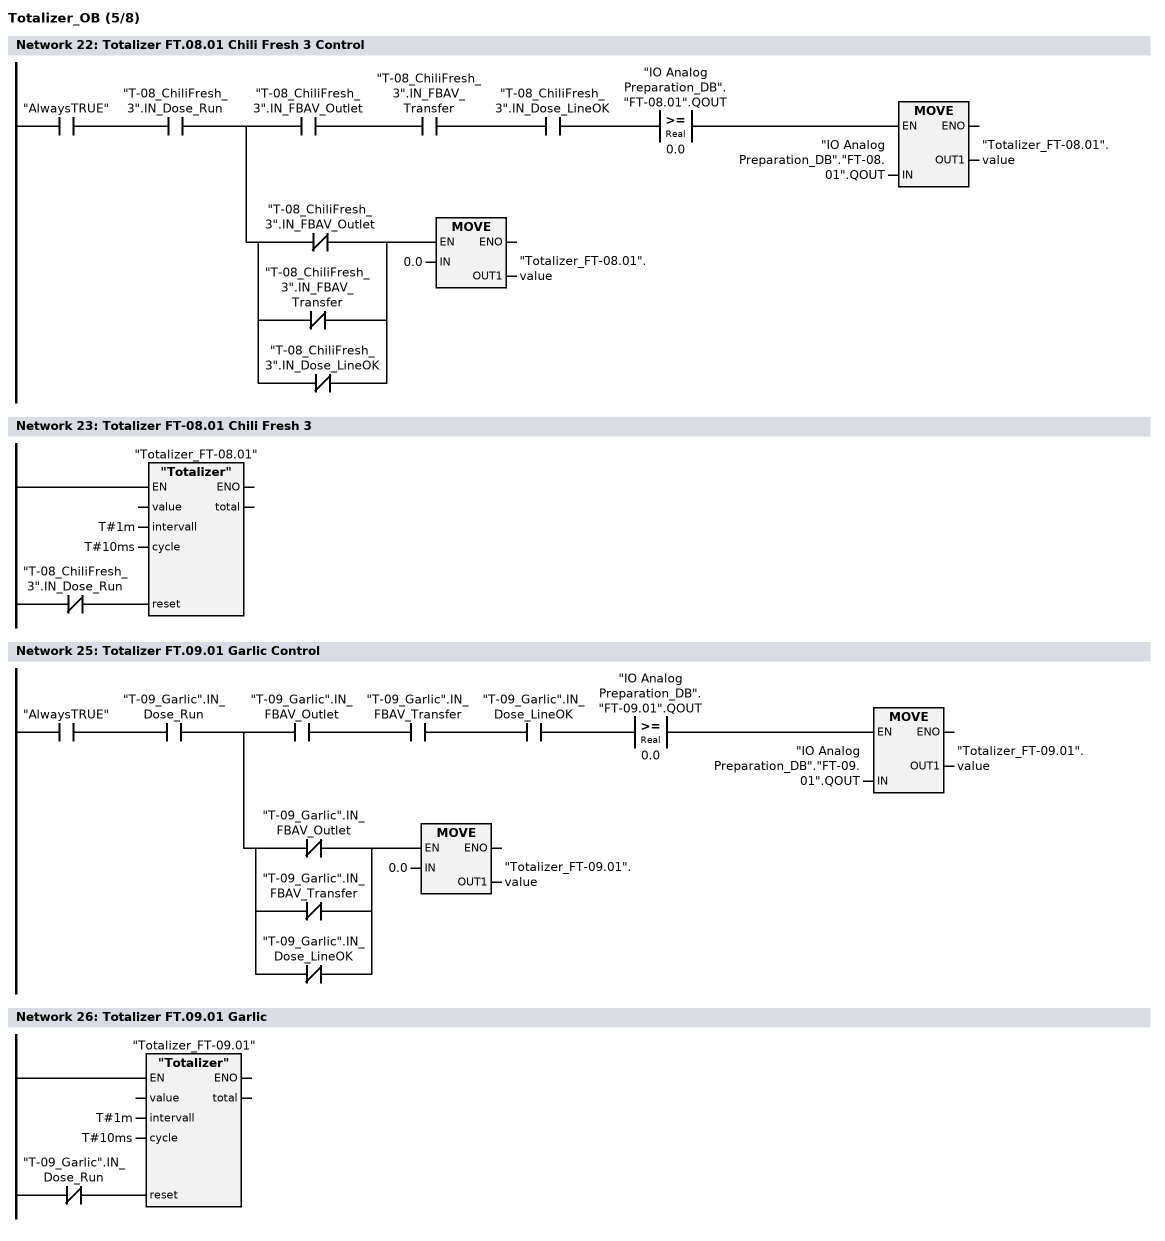
   RUNG wire#powerrail
      Contact( "AlwaysTRUE" )
      Contact( "T-08_ChiliFresh_3".IN_Dose_Run )
      wire#w1
      Contact( "T-08_ChiliFresh_3".IN_FBAV_Outlet )
      Contact( "T-08_ChiliFresh_3".IN_FBAV_Transfer )
      Contact( "T-08_ChiliFresh_3".IN_Dose_LineOK )
      { S7_Templates := "SrcType := Real" } GE_Contact(in1 := "IO Analog Preparation_DB"."FT-08.01".QOUT, in2 := 0.0)
      Move(in := "IO Analog Preparation_DB"."FT-08.01".QOUT, out1 => "Totalizer_FT-08.01".value)
   END_RUNG
   RUNG wire#w1
      I_Contact( "T-08_ChiliFresh_3".IN_FBAV_Outlet )
      wire#w2
      Move(in := 0.0, out1 => "Totalizer_FT-08.01".value)
   END_RUNG
   RUNG wire#w1
      I_Contact( "T-08_ChiliFresh_3".IN_FBAV_Transfer )
   END_RUNG wire#w2
   RUNG wire#w1
      I_Contact( "T-08_ChiliFresh_3".IN_Dose_LineOK )
   END_RUNG wire#w2
   // the same network as SCL:
   #_w1 := "AlwaysTRUE" AND "T-08_ChiliFresh_3".IN_Dose_Run;
   IF #_w1 AND "T-08_ChiliFresh_3".IN_FBAV_Outlet AND "T-08_ChiliFresh_3".IN_FBAV_Transfer AND "T-08_ChiliFresh_3".IN_Dose_LineOK AND ("IO Analog Preparation_DB"."FT-08.01".QOUT >= 0.0) THEN
       "Totalizer_FT-08.01".value := "IO Analog Preparation_DB"."FT-08.01".QOUT;
   END_IF;
   IF #_w1 AND (NOT "T-08_ChiliFresh_3".IN_FBAV_Outlet OR NOT "T-08_ChiliFresh_3".IN_FBAV_Transfer OR NOT "T-08_ChiliFresh_3".IN_Dose_LineOK) THEN
       "Totalizer_FT-08.01".value := 0.0;
   END_IF;
END_REGION

REGION Network 23: Totalizer FT-08.01 Chili Fresh 3
   RUNG wire#powerrail
      "Totalizer_FT-08.01"(reset := wire#w1, value :=, intervall := T#1m, cycle := T#10ms, total =>)
   END_RUNG
   RUNG wire#powerrail
      I_Contact( "T-08_ChiliFresh_3".IN_Dose_Run )
   END_RUNG wire#w1
   // the same network as SCL:
   "Totalizer_FT-08.01"(intervall := T#1m, cycle := T#10ms, reset := NOT "T-08_ChiliFresh_3".IN_Dose_Run);   // "Totalizer"
END_REGION

REGION Network 25: Totalizer FT.09.01 Garlic Control
   RUNG wire#powerrail
      Contact( "AlwaysTRUE" )
      Contact( "T-09_Garlic".IN_Dose_Run )
      wire#w1
      Contact( "T-09_Garlic".IN_FBAV_Outlet )
      Contact( "T-09_Garlic".IN_FBAV_Transfer )
      Contact( "T-09_Garlic".IN_Dose_LineOK )
      { S7_Templates := "SrcType := Real" } GE_Contact(in1 := "IO Analog Preparation_DB"."FT-09.01".QOUT, in2 := 0.0)
      Move(in := "IO Analog Preparation_DB"."FT-09.01".QOUT, out1 => "Totalizer_FT-09.01".value)
   END_RUNG
   RUNG wire#w1
      I_Contact( "T-09_Garlic".IN_FBAV_Outlet )
      wire#w2
      Move(in := 0.0, out1 => "Totalizer_FT-09.01".value)
   END_RUNG
   RUNG wire#w1
      I_Contact( "T-09_Garlic".IN_FBAV_Transfer )
   END_RUNG wire#w2
   RUNG wire#w1
      I_Contact( "T-09_Garlic".IN_Dose_LineOK )
   END_RUNG wire#w2
   // the same network as SCL:
   #_w1 := "AlwaysTRUE" AND "T-09_Garlic".IN_Dose_Run;
   IF #_w1 AND "T-09_Garlic".IN_FBAV_Outlet AND "T-09_Garlic".IN_FBAV_Transfer AND "T-09_Garlic".IN_Dose_LineOK AND ("IO Analog Preparation_DB"."FT-09.01".QOUT >= 0.0) THEN
       "Totalizer_FT-09.01".value := "IO Analog Preparation_DB"."FT-09.01".QOUT;
   END_IF;
   IF #_w1 AND (NOT "T-09_Garlic".IN_FBAV_Outlet OR NOT "T-09_Garlic".IN_FBAV_Transfer OR NOT "T-09_Garlic".IN_Dose_LineOK) THEN
       "Totalizer_FT-09.01".value := 0.0;
   END_IF;
END_REGION

REGION Network 26: Totalizer FT.09.01 Garlic
   RUNG wire#powerrail
      "Totalizer_FT-09.01"(reset := wire#w1, value :=, intervall := T#1m, cycle := T#10ms, total =>)
   END_RUNG
   RUNG wire#powerrail
      I_Contact( "T-09_Garlic".IN_Dose_Run )
   END_RUNG wire#w1
   // the same network as SCL:
   "Totalizer_FT-09.01"(intervall := T#1m, cycle := T#10ms, reset := NOT "T-09_Garlic".IN_Dose_Run);   // "Totalizer"
END_REGION

REGION Network 28: Totalizer FT.10.01 Vinegar Control
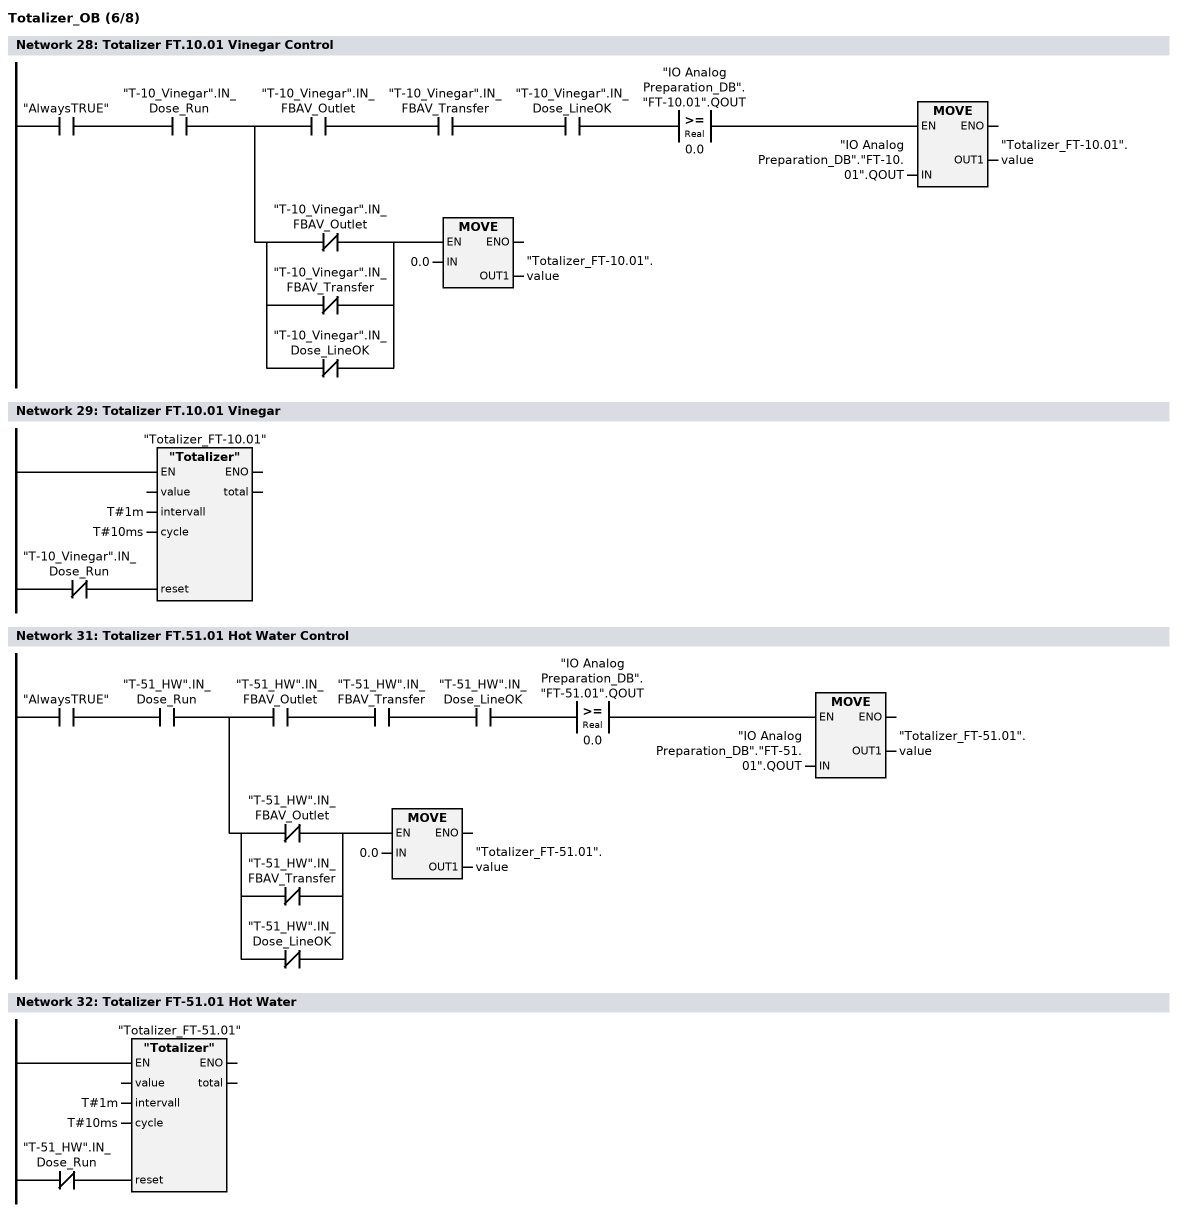
   RUNG wire#powerrail
      Contact( "AlwaysTRUE" )
      Contact( "T-10_Vinegar".IN_Dose_Run )
      wire#w1
      Contact( "T-10_Vinegar".IN_FBAV_Outlet )
      Contact( "T-10_Vinegar".IN_FBAV_Transfer )
      Contact( "T-10_Vinegar".IN_Dose_LineOK )
      { S7_Templates := "SrcType := Real" } GE_Contact(in1 := "IO Analog Preparation_DB"."FT-10.01".QOUT, in2 := 0.0)
      Move(in := "IO Analog Preparation_DB"."FT-10.01".QOUT, out1 => "Totalizer_FT-10.01".value)
   END_RUNG
   RUNG wire#w1
      I_Contact( "T-10_Vinegar".IN_FBAV_Outlet )
      wire#w2
      Move(in := 0.0, out1 => "Totalizer_FT-10.01".value)
   END_RUNG
   RUNG wire#w1
      I_Contact( "T-10_Vinegar".IN_FBAV_Transfer )
   END_RUNG wire#w2
   RUNG wire#w1
      I_Contact( "T-10_Vinegar".IN_Dose_LineOK )
   END_RUNG wire#w2
   // the same network as SCL:
   #_w1 := "AlwaysTRUE" AND "T-10_Vinegar".IN_Dose_Run;
   IF #_w1 AND "T-10_Vinegar".IN_FBAV_Outlet AND "T-10_Vinegar".IN_FBAV_Transfer AND "T-10_Vinegar".IN_Dose_LineOK AND ("IO Analog Preparation_DB"."FT-10.01".QOUT >= 0.0) THEN
       "Totalizer_FT-10.01".value := "IO Analog Preparation_DB"."FT-10.01".QOUT;
   END_IF;
   IF #_w1 AND (NOT "T-10_Vinegar".IN_FBAV_Outlet OR NOT "T-10_Vinegar".IN_FBAV_Transfer OR NOT "T-10_Vinegar".IN_Dose_LineOK) THEN
       "Totalizer_FT-10.01".value := 0.0;
   END_IF;
END_REGION

REGION Network 29: Totalizer FT.10.01 Vinegar
   RUNG wire#powerrail
      "Totalizer_FT-10.01"(reset := wire#w1, value :=, intervall := T#1m, cycle := T#10ms, total =>)
   END_RUNG
   RUNG wire#powerrail
      I_Contact( "T-10_Vinegar".IN_Dose_Run )
   END_RUNG wire#w1
   // the same network as SCL:
   "Totalizer_FT-10.01"(intervall := T#1m, cycle := T#10ms, reset := NOT "T-10_Vinegar".IN_Dose_Run);   // "Totalizer"
END_REGION

REGION Network 31: Totalizer FT.51.01 Hot Water Control
   RUNG wire#powerrail
      Contact( "AlwaysTRUE" )
      Contact( "T-51_HW".IN_Dose_Run )
      wire#w1
      Contact( "T-51_HW".IN_FBAV_Outlet )
      Contact( "T-51_HW".IN_FBAV_Transfer )
      Contact( "T-51_HW".IN_Dose_LineOK )
      { S7_Templates := "SrcType := Real" } GE_Contact(in1 := "IO Analog Preparation_DB"."FT-51.01".QOUT, in2 := 0.0)
      Move(in := "IO Analog Preparation_DB"."FT-51.01".QOUT, out1 => "Totalizer_FT-51.01".value)
   END_RUNG
   RUNG wire#w1
      I_Contact( "T-51_HW".IN_FBAV_Outlet )
      wire#w2
      Move(in := 0.0, out1 => "Totalizer_FT-51.01".value)
   END_RUNG
   RUNG wire#w1
      I_Contact( "T-51_HW".IN_FBAV_Transfer )
   END_RUNG wire#w2
   RUNG wire#w1
      I_Contact( "T-51_HW".IN_Dose_LineOK )
   END_RUNG wire#w2
   // the same network as SCL:
   #_w1 := "AlwaysTRUE" AND "T-51_HW".IN_Dose_Run;
   IF #_w1 AND "T-51_HW".IN_FBAV_Outlet AND "T-51_HW".IN_FBAV_Transfer AND "T-51_HW".IN_Dose_LineOK AND ("IO Analog Preparation_DB"."FT-51.01".QOUT >= 0.0) THEN
       "Totalizer_FT-51.01".value := "IO Analog Preparation_DB"."FT-51.01".QOUT;
   END_IF;
   IF #_w1 AND (NOT "T-51_HW".IN_FBAV_Outlet OR NOT "T-51_HW".IN_FBAV_Transfer OR NOT "T-51_HW".IN_Dose_LineOK) THEN
       "Totalizer_FT-51.01".value := 0.0;
   END_IF;
END_REGION

REGION Network 32: Totalizer FT-51.01 Hot Water
   RUNG wire#powerrail
      "Totalizer_FT-51.01"(reset := wire#w1, value :=, intervall := T#1m, cycle := T#10ms, total =>)
   END_RUNG
   RUNG wire#powerrail
      I_Contact( "T-51_HW".IN_Dose_Run )
   END_RUNG wire#w1
   // the same network as SCL:
   "Totalizer_FT-51.01"(intervall := T#1m, cycle := T#10ms, reset := NOT "T-51_HW".IN_Dose_Run);   // "Totalizer"
END_REGION

REGION Network 34: Totalizer FT-12.01 ProWater Homomixer Control
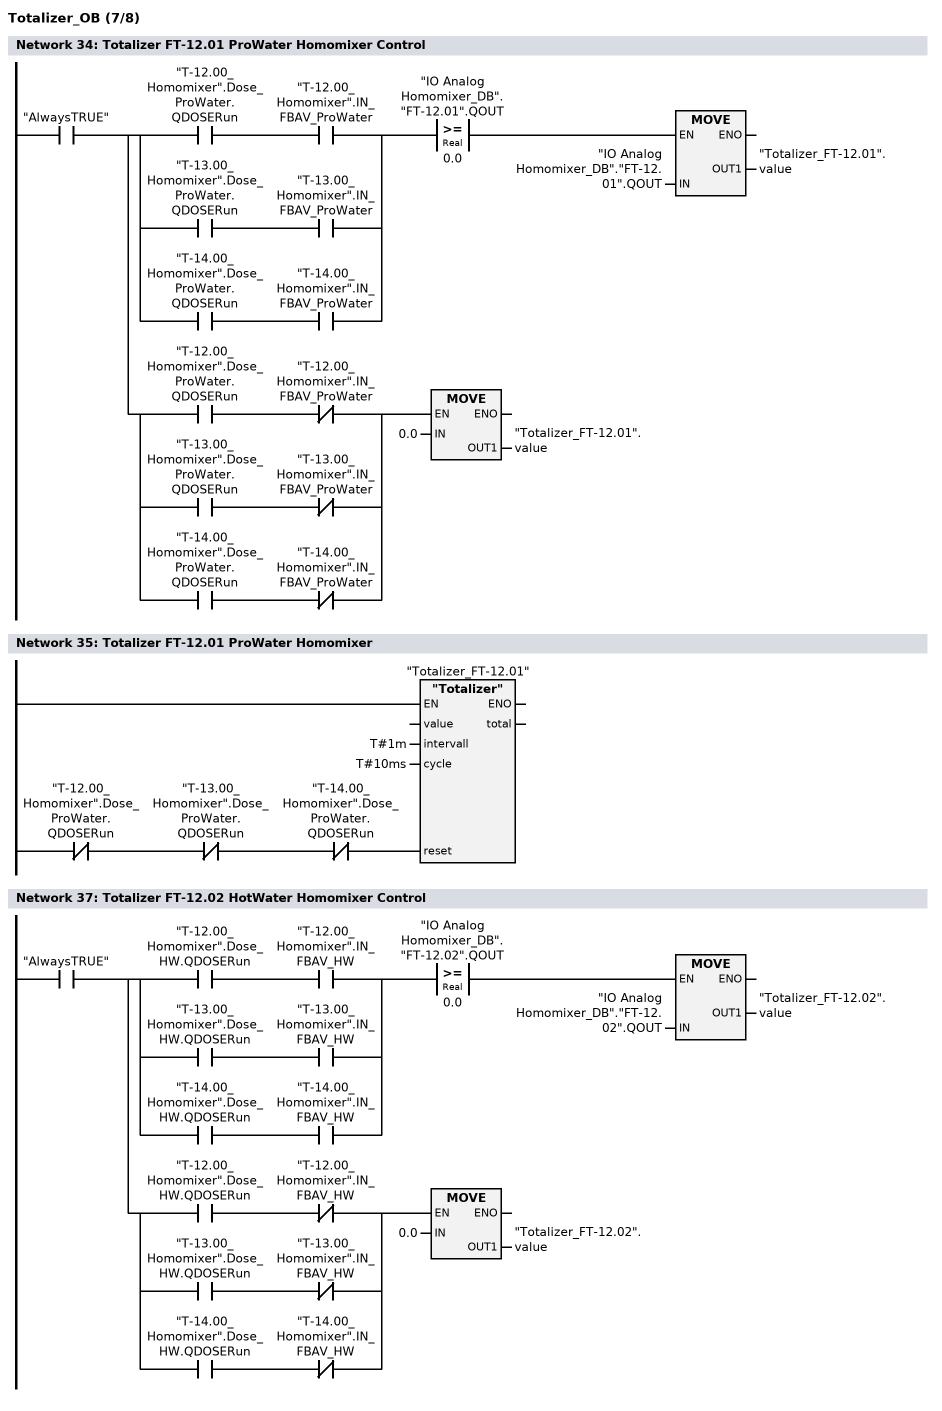
   RUNG wire#powerrail
      Contact( "AlwaysTRUE" )
      wire#w1
      Contact( "T-12.00_Homomixer".Dose_ProWater.QDOSERun )
      Contact( "T-12.00_Homomixer".IN_FBAV_ProWater )
      wire#w2
      { S7_Templates := "SrcType := Real" } GE_Contact(in1 := "IO Analog Homomixer_DB"."FT-12.01".QOUT, in2 := 0.0)
      Move(in := "IO Analog Homomixer_DB"."FT-12.01".QOUT, out1 => "Totalizer_FT-12.01".value)
   END_RUNG
   RUNG wire#w1
      Contact( "T-13.00_Homomixer".Dose_ProWater.QDOSERun )
      Contact( "T-13.00_Homomixer".IN_FBAV_ProWater )
   END_RUNG wire#w2
   RUNG wire#w1
      Contact( "T-14.00_Homomixer".Dose_ProWater.QDOSERun )
      Contact( "T-14.00_Homomixer".IN_FBAV_ProWater )
   END_RUNG wire#w2
   RUNG wire#w1
      Contact( "T-12.00_Homomixer".Dose_ProWater.QDOSERun )
      I_Contact( "T-12.00_Homomixer".IN_FBAV_ProWater )
      wire#w3
      Move(in := 0.0, out1 => "Totalizer_FT-12.01".value)
   END_RUNG
   RUNG wire#w1
      Contact( "T-13.00_Homomixer".Dose_ProWater.QDOSERun )
      I_Contact( "T-13.00_Homomixer".IN_FBAV_ProWater )
   END_RUNG wire#w3
   RUNG wire#w1
      Contact( "T-14.00_Homomixer".Dose_ProWater.QDOSERun )
      I_Contact( "T-14.00_Homomixer".IN_FBAV_ProWater )
   END_RUNG wire#w3
   // the same network as SCL:
   IF "AlwaysTRUE" AND (("T-12.00_Homomixer".Dose_ProWater.QDOSERun AND "T-12.00_Homomixer".IN_FBAV_ProWater) OR ("T-13.00_Homomixer".Dose_ProWater.QDOSERun AND "T-13.00_Homomixer".IN_FBAV_ProWater) OR ("T-14.00_Homomixer".Dose_ProWater.QDOSERun AND "T-14.00_Homomixer".IN_FBAV_ProWater)) AND ("IO Analog Homomixer_DB"."FT-12.01".QOUT >= 0.0) THEN
       "Totalizer_FT-12.01".value := "IO Analog Homomixer_DB"."FT-12.01".QOUT;
   END_IF;
   IF "AlwaysTRUE" AND (("T-12.00_Homomixer".Dose_ProWater.QDOSERun AND NOT "T-12.00_Homomixer".IN_FBAV_ProWater) OR ("T-13.00_Homomixer".Dose_ProWater.QDOSERun AND NOT "T-13.00_Homomixer".IN_FBAV_ProWater) OR ("T-14.00_Homomixer".Dose_ProWater.QDOSERun AND NOT "T-14.00_Homomixer".IN_FBAV_ProWater)) THEN
       "Totalizer_FT-12.01".value := 0.0;
   END_IF;
END_REGION

REGION Network 35: Totalizer FT-12.01 ProWater Homomixer
   RUNG wire#powerrail
      "Totalizer_FT-12.01"(reset := wire#w1, value :=, intervall := T#1m, cycle := T#10ms, total =>)
   END_RUNG
   RUNG wire#powerrail
      I_Contact( "T-12.00_Homomixer".Dose_ProWater.QDOSERun )
      I_Contact( "T-13.00_Homomixer".Dose_ProWater.QDOSERun )
      I_Contact( "T-14.00_Homomixer".Dose_ProWater.QDOSERun )
   END_RUNG wire#w1
   // the same network as SCL:
   "Totalizer_FT-12.01"(intervall := T#1m,   // "Totalizer"
                        cycle := T#10ms,
                        reset := NOT "T-12.00_Homomixer".Dose_ProWater.QDOSERun AND NOT "T-13.00_Homomixer".Dose_ProWater.QDOSERun AND NOT "T-14.00_Homomixer".Dose_ProWater.QDOSERun);
END_REGION

REGION Network 37: Totalizer FT-12.02 HotWater Homomixer Control
   RUNG wire#powerrail
      Contact( "AlwaysTRUE" )
      wire#w1
      Contact( "T-12.00_Homomixer".Dose_HW.QDOSERun )
      Contact( "T-12.00_Homomixer".IN_FBAV_HW )
      wire#w2
      { S7_Templates := "SrcType := Real" } GE_Contact(in1 := "IO Analog Homomixer_DB"."FT-12.02".QOUT, in2 := 0.0)
      Move(in := "IO Analog Homomixer_DB"."FT-12.02".QOUT, out1 => "Totalizer_FT-12.02".value)
   END_RUNG
   RUNG wire#w1
      Contact( "T-13.00_Homomixer".Dose_HW.QDOSERun )
      Contact( "T-13.00_Homomixer".IN_FBAV_HW )
   END_RUNG wire#w2
   RUNG wire#w1
      Contact( "T-14.00_Homomixer".Dose_HW.QDOSERun )
      Contact( "T-14.00_Homomixer".IN_FBAV_HW )
   END_RUNG wire#w2
   RUNG wire#w1
      Contact( "T-12.00_Homomixer".Dose_HW.QDOSERun )
      I_Contact( "T-12.00_Homomixer".IN_FBAV_HW )
      wire#w3
      Move(in := 0.0, out1 => "Totalizer_FT-12.02".value)
   END_RUNG
   RUNG wire#w1
      Contact( "T-13.00_Homomixer".Dose_HW.QDOSERun )
      I_Contact( "T-13.00_Homomixer".IN_FBAV_HW )
   END_RUNG wire#w3
   RUNG wire#w1
      Contact( "T-14.00_Homomixer".Dose_HW.QDOSERun )
      I_Contact( "T-14.00_Homomixer".IN_FBAV_HW )
   END_RUNG wire#w3
   // the same network as SCL:
   IF "AlwaysTRUE" AND (("T-12.00_Homomixer".Dose_HW.QDOSERun AND "T-12.00_Homomixer".IN_FBAV_HW) OR ("T-13.00_Homomixer".Dose_HW.QDOSERun AND "T-13.00_Homomixer".IN_FBAV_HW) OR ("T-14.00_Homomixer".Dose_HW.QDOSERun AND "T-14.00_Homomixer".IN_FBAV_HW)) AND ("IO Analog Homomixer_DB"."FT-12.02".QOUT >= 0.0) THEN
       "Totalizer_FT-12.02".value := "IO Analog Homomixer_DB"."FT-12.02".QOUT;
   END_IF;
   IF "AlwaysTRUE" AND (("T-12.00_Homomixer".Dose_HW.QDOSERun AND NOT "T-12.00_Homomixer".IN_FBAV_HW) OR ("T-13.00_Homomixer".Dose_HW.QDOSERun AND NOT "T-13.00_Homomixer".IN_FBAV_HW) OR ("T-14.00_Homomixer".Dose_HW.QDOSERun AND NOT "T-14.00_Homomixer".IN_FBAV_HW)) THEN
       "Totalizer_FT-12.02".value := 0.0;
   END_IF;
END_REGION

REGION Network 38: Totalizer FT-12.02 HotWater Homomixer
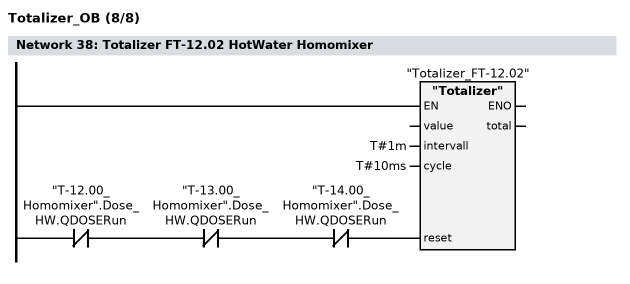
   RUNG wire#powerrail
      "Totalizer_FT-12.02"(reset := wire#w1, value :=, intervall := T#1m, cycle := T#10ms, total =>)
   END_RUNG
   RUNG wire#powerrail
      I_Contact( "T-12.00_Homomixer".Dose_HW.QDOSERun )
      I_Contact( "T-13.00_Homomixer".Dose_HW.QDOSERun )
      I_Contact( "T-14.00_Homomixer".Dose_HW.QDOSERun )
   END_RUNG wire#w1
   // the same network as SCL:
   "Totalizer_FT-12.02"(intervall := T#1m,   // "Totalizer"
                        cycle := T#10ms,
                        reset := NOT "T-12.00_Homomixer".Dose_HW.QDOSERun AND NOT "T-13.00_Homomixer".Dose_HW.QDOSERun AND NOT "T-14.00_Homomixer".Dose_HW.QDOSERun);
END_REGION
END_ORGANIZATION_BLOCK

FUNCTION_BLOCK "Totalizer"
{ S7_Optimized_Access := 'TRUE' }
VERSION : 0.1
   VAR_INPUT 
      value : Real;
      intervall : Time;
      cycle : Time;
      reset : Bool;
   END_VAR

   VAR_OUTPUT 
      total : Real;
   END_VAR

   VAR 
      statAccum : Real;
   END_VAR

   VAR_TEMP 
      tempIntervall : Real;
      tempCycle : Real;
      tempIntervallDInt : DInt;
      tempCycleDInt : DInt;
   END_VAR


BEGIN
	//Ist der Signalzustand der Variable "Reset" gleich True, so werden die Variablen
	//"Accum" und "Total" auf Null zurückgesetzt und es erfolgt keine Berechnung.
	//Beim Signalzustand False erfolgt zunächst eine Datentypumwandlung nach Real der beiden
	//Eingangsvariablen "Intervall" und "Cycle". Zuerst mit der Konvertierung von Time nach
	//DInt und anschließend von DInt nach Real.
	//Innerhalb eines Zyklus wird der Eingangswert der Variablen "Value" mit dem Wert der temporären Variablen
	//"Cycle_real" multipliziert und mit dem Wert der temporären Variablen "Intervall_real" dividiert.
	//Das Ergebnis wird anschließend in den Zwischenspeicher "Accum" abgelegt. Somit wird innerhalb eines jeden
	//Zykluses das Zwischenergebnis im "Accum" um diesen Wert inkrementiert, welches auch in jedem Zyklus zur
	//Ausgangsvariable "Total" transferiert wird.
	//***************************************************************************
	//If the signal status of the variable "Reset" is true, the variables "Accum" and "Total"
	//are set to zero and there is no calculation.
	//If the signal status is false, there is first a data type change to real of the two
	//input variables "Intervall" and "Cycle. After conversion from Time to DInit and from DInt to Real.
	//In a #Cycle the input #Value of the variable "Value" is multiplied by the #Value of the temporary variable
	//"Cycle_real" and then divided by the #Value of the temporary variable "Intervall_real". The result is then
	//stored in the buffer "Accum". This in one particular #Cycle the result in the "Accum" buffer is
	//incremented this #Value, which is also transferred to the output variable "Total" in that #Cycle too.
	
	IF #reset = true THEN
	    #statAccum := 0.000000e000; //Die Variablen werden zurückgesetzt.
	    #total := 0.000000e000; //The variables will be set to zero.
	ELSE
	    #tempIntervallDInt := TIME_TO_DINT(#intervall);
	    #tempIntervall := DINT_TO_REAL(#tempIntervallDInt);
	    #tempCycleDInt := TIME_TO_DINT(#cycle);
	    #tempCycle := DINT_TO_REAL(#tempCycleDInt);
	    #statAccum := ((#value * #tempCycle) / #tempIntervall) + #statAccum;
	    #total := #statAccum; //Kopiere Ergebnis nach #Total / Copy result to #Total.
	END_IF;
END_FUNCTION_BLOCK

FUNCTION "Transfer_Homomix" : Void   // FC9, LAD
{ S7_Optimized_Access := 'TRUE' }
VERSION : 0.1
// stored: AutoNumber true, IsIECCheckEnabled false, SetENOAutomatically false, UDAEnableTagReadback false
   VAR_INPUT
      req : Bool;
      "low level" : Bool;
      "tank inload" : Bool;
      "cmd start" : Bool;
      "cmd stop" : Bool;
      "FB AV Transfer" : Bool;
      "FB SV Pump" : Bool;
   END_VAR
   VAR_OUTPUT
      "AV Transfer" : Bool;
      "SV Pump" : Bool;
      indicator_start : Bool;
      indicator_stop : Bool;
   END_VAR
   VAR_IN_OUT
      "cmd en start" : Bool;
      "cmd en stop" : Bool;
      "cmd state start" : Bool;
      "cmd state stop" : Bool;
      indicator_request : Bool;
      "always ON" : Bool;
   END_VAR
   VAR_TEMP   // added for the SCL form of the ladder/FBD networks
      _w1 : Bool;
      _w2 : Bool;
   END_VAR
BEGIN

REGION Network 1
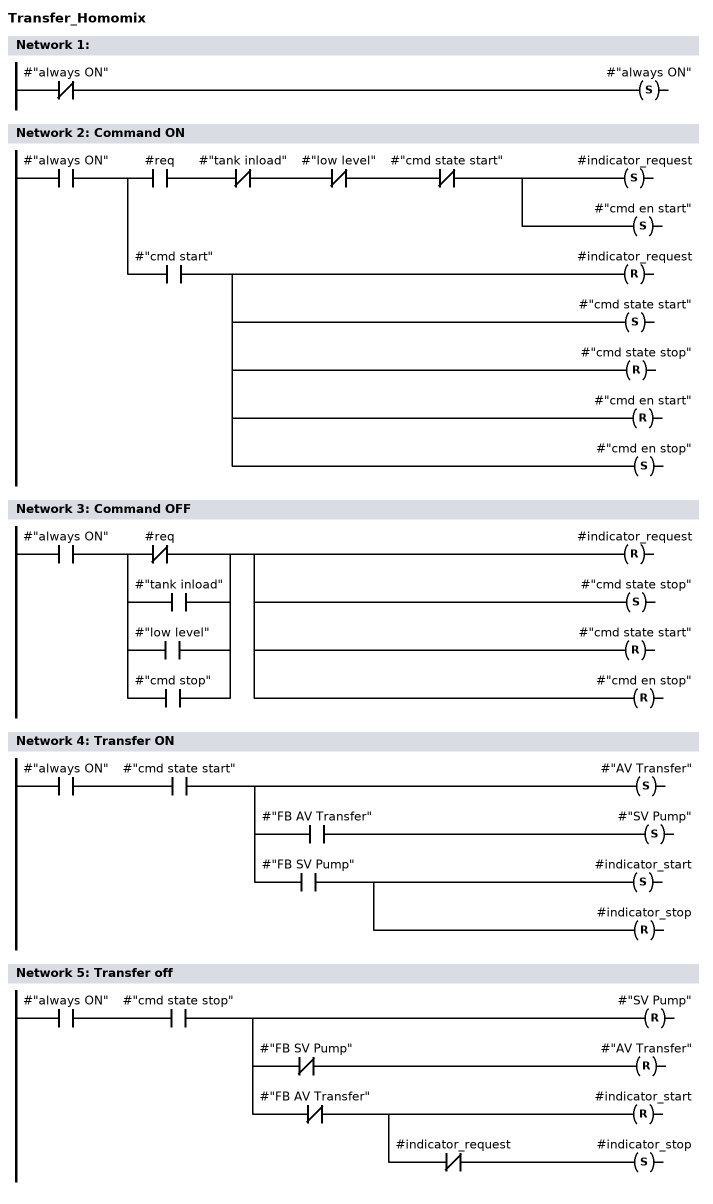
   RUNG wire#powerrail
      I_Contact( #"always ON" )
      S_Coil( #"always ON" )
   END_RUNG
   // the same network as SCL:
   IF NOT #"always ON" THEN #"always ON" := TRUE; END_IF;
END_REGION

REGION Network 2: Command ON
   RUNG wire#powerrail
      Contact( #"always ON" )
      wire#w1
      Contact( #req )
      I_Contact( #"tank inload" )
      I_Contact( #"low level" )
      I_Contact( #"cmd state start" )
      wire#w2
      S_Coil( #indicator_request )
   END_RUNG
   RUNG wire#w2
      S_Coil( #"cmd en start" )
   END_RUNG
   RUNG wire#w1
      Contact( #"cmd start" )
      wire#w3
      R_Coil( #indicator_request )
   END_RUNG
   RUNG wire#w3
      S_Coil( #"cmd state start" )
   END_RUNG
   RUNG wire#w3
      R_Coil( #"cmd state stop" )
   END_RUNG
   RUNG wire#w3
      R_Coil( #"cmd en start" )
   END_RUNG
   RUNG wire#w3
      S_Coil( #"cmd en stop" )
   END_RUNG
   // the same network as SCL:
   IF #"always ON" AND #req AND NOT #"tank inload" AND NOT #"low level" AND NOT #"cmd state start" THEN
       #indicator_request := TRUE;
       #"cmd en start" := TRUE;
   END_IF;
   IF #"always ON" AND #"cmd start" THEN
       #indicator_request := FALSE;
       #"cmd state start" := TRUE;
       #"cmd state stop" := FALSE;
       #"cmd en start" := FALSE;
       #"cmd en stop" := TRUE;
   END_IF;
END_REGION

REGION Network 3: Command OFF
   RUNG wire#powerrail
      Contact( #"always ON" )
      wire#w1
      I_Contact( #req )
      wire#w2
      R_Coil( #indicator_request )
   END_RUNG
   RUNG wire#w1
      Contact( #"tank inload" )
   END_RUNG wire#w2
   RUNG wire#w1
      Contact( #"low level" )
   END_RUNG wire#w2
   RUNG wire#w1
      Contact( #"cmd stop" )
   END_RUNG wire#w2
   RUNG wire#w2
      S_Coil( #"cmd state stop" )
   END_RUNG
   RUNG wire#w2
      R_Coil( #"cmd state start" )
   END_RUNG
   RUNG wire#w2
      R_Coil( #"cmd en stop" )
   END_RUNG
   // the same network as SCL:
   IF #"always ON" AND (NOT #req OR #"tank inload" OR #"low level" OR #"cmd stop") THEN
       #indicator_request := FALSE;
       #"cmd state stop" := TRUE;
       #"cmd state start" := FALSE;
       #"cmd en stop" := FALSE;
   END_IF;
END_REGION

REGION Network 4: Transfer ON
   RUNG wire#powerrail
      Contact( #"always ON" )
      Contact( #"cmd state start" )
      wire#w1
      S_Coil( #"AV Transfer" )
   END_RUNG
   RUNG wire#w1
      Contact( #"FB AV Transfer" )
      S_Coil( #"SV Pump" )
   END_RUNG
   RUNG wire#w1
      Contact( #"FB SV Pump" )
      wire#w2
      S_Coil( #indicator_start )
   END_RUNG
   RUNG wire#w2
      R_Coil( #indicator_stop )
   END_RUNG
   // the same network as SCL:
   #_w1 := #"always ON" AND #"cmd state start";
   IF #_w1 THEN #"AV Transfer" := TRUE; END_IF;
   IF #_w1 AND #"FB AV Transfer" THEN #"SV Pump" := TRUE; END_IF;
   IF #_w1 AND #"FB SV Pump" THEN
       #indicator_start := TRUE;
       #indicator_stop := FALSE;
   END_IF;
END_REGION

REGION Network 5: Transfer off
   RUNG wire#powerrail
      Contact( #"always ON" )
      Contact( #"cmd state stop" )
      wire#w1
      R_Coil( #"SV Pump" )
   END_RUNG
   RUNG wire#w1
      I_Contact( #"FB SV Pump" )
      R_Coil( #"AV Transfer" )
   END_RUNG
   RUNG wire#w1
      I_Contact( #"FB AV Transfer" )
      wire#w2
      R_Coil( #indicator_start )
   END_RUNG
   RUNG wire#w2
      I_Contact( #indicator_request )
      S_Coil( #indicator_stop )
   END_RUNG
   // the same network as SCL:
   #_w1 := #"always ON" AND #"cmd state stop";
   IF #_w1 THEN #"SV Pump" := FALSE; END_IF;
   IF #_w1 AND NOT #"FB SV Pump" THEN #"AV Transfer" := FALSE; END_IF;
   #_w2 := #_w1 AND NOT #"FB AV Transfer";
   IF #_w2 THEN #indicator_start := FALSE; END_IF;
   IF #_w2 AND NOT #indicator_request THEN #indicator_stop := TRUE; END_IF;
END_REGION
END_FUNCTION

FUNCTION_BLOCK "Danfos_VSD"   // FB623, LAD
{ S7_Optimized_Access := 'FALSE' }
VERSION : 0.1
// stored: AutoNumber false, IsIECCheckEnabled false, SetENOAutomatically false, UDAEnableTagReadback false
   VAR_INPUT
      In_CMD : Bool;   // 0 = Stop, 1 = Start
      Reset : Bool;
      QuickStop : Bool;   // 1 = Emergency stop
      drive_f_setpoint : Real;   // Frequency setpoint in Hz; 0.00<f_setl<50.00Hz
      In_STW : Word;
      drive_AV { ExternalAccessible := 'False'; ExternalVisible := 'False'; ExternalWritable := 'False'} : Int;   // Drive Actual value
   END_VAR
   VAR_OUTPUT
      Danfos_CTW : Word;
      Danfos_SP { ExternalAccessible := 'False'; ExternalVisible := 'False'; ExternalWritable := 'False'} : Word;   // Drive Settpoint
      Drive_OK : Bool;
      Drive_Run : Bool;
      QAlarm : Word;
      Danfos_f_act : Real;   // actual_frequency 0...50Hz
      "Danfos_QAV_%" : Real;   // actual_frequency 0..100%
   END_VAR
   VAR DB_SPECIFIC
      SW : Struct
         "Bit 0-Control" : Bool;   // 0 = Control not ready, 1 = Control ready
         "Bit 1-Drive" : Bool;   // 0 = Drive not ready, 1 = Drive ready
         "Bit 2-Coasting stop" : Bool;   // 0 = can't start the motor, 1 = can start the motor
         "Bit 3-Trip" : Bool;   // 0 = No error, 1 = Trip
         "Bit 4-Error" : Bool;   // 0 = No error, 1 = Drive Error (no Trip)
         "Bit 5-NOP" : Bool;
         "Bit 6-triplock" : Bool;   // 0 = not in fault, 1 = tripped and locked
         "Bit 7-Warning" : Bool;   // 0 = No warning , 1 = Warning
         "Bit 8-Speed reference" : Bool;   // 0 = Speed =/ reference, 1 = Speed = reference
         "Bit 9-Operation" : Bool;   // 0 = Local operation, 1 = bus control
         "Bit 10-frequency range" : Bool;   // 0 = Outside frequency range, 1 =Within frequency range
         "Bit 11-Operation" : Bool;   // 0 = No operation, 1 = In operation
         "Bit 12-Drive OK" : Bool;   // 0 = Drive OK, 1 = Stopped, autostart
         "Bit 13-Voltage OK" : Bool;   // 0 = Voltage OK, 1 = Voltage exceeded
         "Bit 14-Torque OK" : Bool;   // 0 = Torque OK, 1 = Torque exceeded
         "Bit 15-Timers OK" : Bool;   // 0 = Timers OK, 1 = Timers exceeded
      END_STRUCT;
      Reset_PE : Bool;
      Reset_Bits : Bool;
      f_act : Real;
   END_VAR
   VAR_TEMP   // added for the SCL form of the ladder/FBD networks
      _w1 : Bool;
   END_VAR
BEGIN

REGION Network 1: Reset
   // Bit Bit value=0 Bit value=1
   // 00 Reference value External selection lsb
   // 01 Reference value External selection msb
   // 02 DC brake Ramp
   // 03 Coasting No coasting
   // 04 Quick stop Ramp
   // 05 Hold output frequency Use ramp
   // 06 Ramp stop Start
   // 07 No function Reset
   // 08 No function Jog
   // 09 Ramp 1 Ramp 2
   // 10 Data invalid Data valid
   // 11 No function Relay 01 active
   // 12 No function Relay 04 active
   // 13 Parameter set-up selection lsb
   // 14 Parameter set-up selection msb
   // 15 No function Reverse
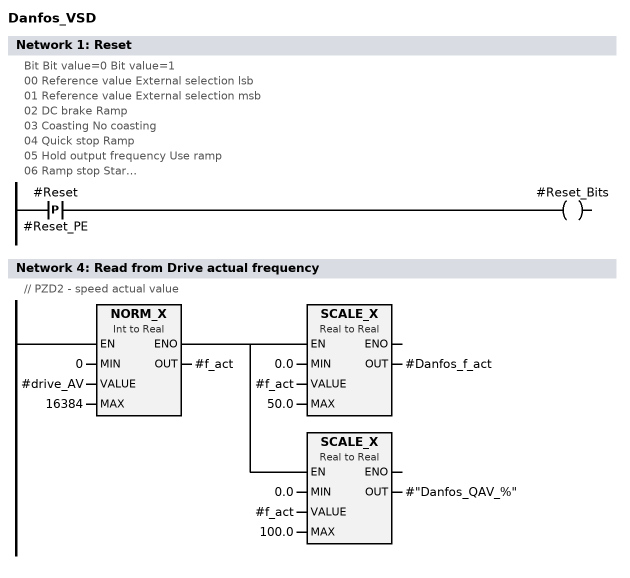
   RUNG wire#powerrail
      P_Contact(operand := #Reset, bit := #Reset_PE)
      Coil( #Reset_Bits )
   END_RUNG
   // the same network as SCL:
   #_w1 := #Reset AND NOT #Reset_PE;   // rising edge of #Reset
   #Reset_PE := #Reset;
   #Reset_Bits := #_w1;
END_REGION

REGION Network 2 (SCL): Read Status Word
   #SW."Bit 0-Control" := #In_STW.%X0;
   #SW."Bit 1-Drive" := #In_STW.%X1;
   #SW."Bit 2-Coasting stop" := #In_STW.%X2;
   #SW."Bit 3-Trip" := #In_STW.%X3;
   #SW."Bit 4-Error" := #In_STW.%X4;
   #SW."Bit 5-NOP" := #In_STW.%X5;
   #SW."Bit 6-triplock" := #In_STW.%X6;
   #SW."Bit 7-Warning" := #In_STW.%X7;
   #SW."Bit 8-Speed reference" := #In_STW.%X8;
   #SW."Bit 9-Operation" := #In_STW.%X9;
   #SW."Bit 10-frequency range" := #In_STW.%X10;
   #SW."Bit 11-Operation" := #In_STW.%X11;
   #SW."Bit 12-Drive OK" := #In_STW.%X12;
   #SW."Bit 13-Voltage OK" := #In_STW.%X13;
   #SW."Bit 14-Torque OK" := #In_STW.%X14;
   #SW."Bit 15-Timers OK" := #In_STW.%X15;
END_REGION

REGION Network 3 (SCL): Drive Status
   #Drive_Run := #SW."Bit 11-Operation" = true;

   #Drive_OK := (#SW."Bit 0-Control" = true AND
                 #SW."Bit 1-Drive" = true ) OR
                 (#SW."Bit 2-Coasting stop" = true AND
                 #SW."Bit 3-Trip" = false AND
                 #SW."Bit 4-Error" = false AND
                 #SW."Bit 6-triplock" = false AND
                 #SW."Bit 7-Warning" = false);
END_REGION

REGION Network 4: Read from Drive actual frequency
   // // PZD2 - speed actual value
   RUNG wire#powerrail
      { S7_Templates := "[SrcType := Int, DestType := Real]" } Normalize(min := 0, value := #drive_AV, max := 16384, out => #f_act)
      wire#w1
      { S7_Templates := "[SrcType := Real, DestType := Real]" } Scale(min := 0.0, value := #f_act, max := 50.0, out => #Danfos_f_act)
   END_RUNG
   RUNG wire#w1
      { S7_Templates := "[SrcType := Real, DestType := Real]" } Scale(min := 0.0, value := #f_act, max := 100.0, out => #"Danfos_QAV_%")
   END_RUNG
   // the same network as SCL:
   #f_act := NORM_X(MIN := 0, VALUE := #drive_AV, MAX := 16384);
   #Danfos_f_act := SCALE_X(MIN := 0.0, VALUE := #f_act, MAX := 50.0);
   #"Danfos_QAV_%" := SCALE_X(MIN := 0.0, VALUE := #f_act, MAX := 100.0);
END_REGION

REGION Network 5 (SCL): Write to Drive Control Word
   #Danfos_CTW.%X0 := false;
   #Danfos_CTW.%X1 := false;
   #Danfos_CTW.%X2 := true;
   #Danfos_CTW.%X3 := true;
   #Danfos_CTW.%X4 := #QuickStop = true;
   #Danfos_CTW.%X5 := true;
   #Danfos_CTW.%X6 := (#Drive_OK =true AND #In_CMD =true AND #QuickStop = true);
   #Danfos_CTW.%X7 := #Reset_Bits;
   #Danfos_CTW.%X8 := false;
   #Danfos_CTW.%X9 := false;
   #Danfos_CTW.%X10 := true;
   #Danfos_CTW.%X11 := false;
   #Danfos_CTW.%X12 := false;
   #Danfos_CTW.%X13 := false;
   #Danfos_CTW.%X14 := false;
   #Danfos_CTW.%X15 := false;
END_REGION

NETWORK
TITLE = Write to Drive Setpoint
// PZD2 - speed setpoint
// Valid speed setpoint between 0.00-50.00 Hz

      L     #drive_f_setpoint;  // Load the frequency setpoint [Hz]
      L     0.0;  // Load the value 0
      <R;  // Compare the speed setpoint with 0 (Hz): < 0 Hz ?
      JC    N004;  // Yes: Jump to mark N004; No: Continue program run

      L     #drive_f_setpoint;  // Load the frequency setpoint [Hz]
      L     50.0;  // Load the value 50
      >R;  // Compare the speed setpoint with 50 (Hz): > 50 Hz ?
      JC    N004;  // Yes: Jump to the mark N004; No: Continue program run

      L     #drive_f_setpoint;  // Load the frequency setpoint [Hz]

// Save 2 decimal places:
      L     100.0;  // Load the value 100
      *R;  // Multiply the values
      RND;  // Round-off the value (floating point number) to an integer number
      L     16384;  // Load the value 16384 = 4000HEX = 50Hz
      *D;  // Multiply the values
      L     5000;  // The load the value 5000
      /D;  // Divide the contents of AKKU2 by the contents of AKKU1
      T     #Danfos_SP;  // Transfer to the drive

N004: NOP   0;  // Jump mark N004: No function

END_FUNCTION_BLOCK

FUNCTION_BLOCK "InletWater"   // FB30, LAD
{ S7_Optimized_Access := 'TRUE' }
VERSION : 0.1
// stored: AutoNumber false, IsIECCheckEnabled false, IsRetainMemResEnabled false, MemoryReserve 100, SetENOAutomatically false, UDAEnableTagReadback false
   VAR_INPUT
      IN_FBAV_ProWater : Bool;
      IN_FBAV_HotWater : Bool;
      IN_FBAV_HWT : Bool;
      IN_FT_01 : Real;
      IN_FT_02 : Real;
      IN_FB_PumpHWT : Bool;
   END_VAR
   VAR_OUTPUT
      Q_AV_ProWater : Bool;
      Q_AV_HotWater : Bool;
      Q_PumpHWT : Bool;
   END_VAR
   VAR
      alwaysON : Bool;
      Cmd : Struct
         Pro_Start_Process : Bool;
         Hot_Start_Process : Bool;
         Stop_Process : Bool;
         Reset : Bool;
      END_STRUCT;
      Parameter : Struct
         SP_Prowater : Real;
         SP_Hotwater : Real;
      END_STRUCT;
      State : Struct
         Tank : Struct
            ProWater : Struct
               Idle : Bool;
               Ready_for_Inlet : Bool;
               OnGoing : Bool;
               Error : Bool;
               Done : Bool;
            END_STRUCT;
            HotWater : Struct
               Idle : Bool;
               Ready_for_Inlet : Bool;
               OnGoing : Bool;
               Error : Bool;
               Done : Bool;
            END_STRUCT;
            Status : USInt;
         END_STRUCT;
         HW_Error : Bool;
         Inlet_Done : Bool;
      END_STRUCT;
      Actuator : Struct
         AV_ProWater : Bool;
         AV_HotWater : Bool;
         Pump_HWT : Bool;
      END_STRUCT;
      "Timer" : Struct
         HotWater : IEC_TIMER;
         AVHotWater { S7_SetPoint := 'True'} : IEC_TIMER;
      END_STRUCT;
      N_InletProOnGoing : Bool;
      N_InletHotOnGoing : Bool;
      N_PumpHWT : Bool;
      P_InletProDone : Bool;
      P_InletHotDone : Bool;
      P_Stop : Bool;
      P_Reset : Bool;
      P_InletProReady : Bool;
      N_InletOnGoing : Bool;
   END_VAR
   VAR_TEMP   // added for the SCL form of the ladder/FBD networks
      _w1 : Bool;
      _w2 : Bool;
   END_VAR
BEGIN

REGION Network 1: Always ON
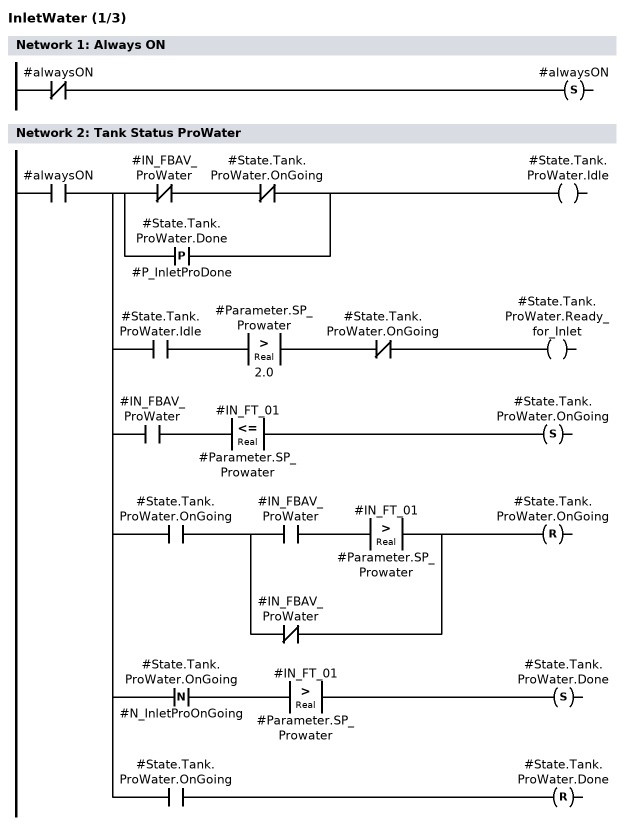
   RUNG wire#powerrail
      I_Contact( #alwaysON )
      S_Coil( #alwaysON )
   END_RUNG
   // the same network as SCL:
   IF NOT #alwaysON THEN #alwaysON := TRUE; END_IF;
END_REGION

REGION Network 2: Tank Status ProWater
   RUNG wire#powerrail
      Contact( #alwaysON )
      wire#w1
      I_Contact( #IN_FBAV_ProWater )
      I_Contact( #State.Tank.ProWater.OnGoing )
      wire#w2
      Coil( #State.Tank.ProWater.Idle )
   END_RUNG
   RUNG wire#w1
      P_Contact(operand := #State.Tank.ProWater.Done, bit := #P_InletProDone)
   END_RUNG wire#w2
   RUNG wire#w1
      Contact( #State.Tank.ProWater.Idle )
      { S7_Templates := "SrcType := Real" } GT_Contact(in1 := #Parameter.SP_Prowater, in2 := 2.0)
      I_Contact( #State.Tank.ProWater.OnGoing )
      Coil( #State.Tank.ProWater.Ready_for_Inlet )
   END_RUNG
   RUNG wire#w1
      Contact( #IN_FBAV_ProWater )
      { S7_Templates := "SrcType := Real" } LE_Contact(in1 := #IN_FT_01, in2 := #Parameter.SP_Prowater)
      S_Coil( #State.Tank.ProWater.OnGoing )
   END_RUNG
   RUNG wire#w1
      Contact( #State.Tank.ProWater.OnGoing )
      wire#w3
      Contact( #IN_FBAV_ProWater )
      { S7_Templates := "SrcType := Real" } GT_Contact(in1 := #IN_FT_01, in2 := #Parameter.SP_Prowater)
      wire#w4
      R_Coil( #State.Tank.ProWater.OnGoing )
   END_RUNG
   RUNG wire#w3
      I_Contact( #IN_FBAV_ProWater )
   END_RUNG wire#w4
   RUNG wire#w1
      N_Contact(operand := #State.Tank.ProWater.OnGoing, bit := #N_InletProOnGoing)
      { S7_Templates := "SrcType := Real" } GT_Contact(in1 := #IN_FT_01, in2 := #Parameter.SP_Prowater)
      S_Coil( #State.Tank.ProWater.Done )
   END_RUNG
   RUNG wire#w1
      Contact( #State.Tank.ProWater.OnGoing )
      R_Coil( #State.Tank.ProWater.Done )
   END_RUNG
   // the same network as SCL:
   #_w1 := #alwaysON AND #State.Tank.ProWater.Done AND NOT #P_InletProDone;   // rising edge of #State.Tank.ProWater.Done
   #P_InletProDone := #State.Tank.ProWater.Done;
   #State.Tank.ProWater.Idle := (#alwaysON AND NOT #IN_FBAV_ProWater AND NOT #State.Tank.ProWater.OnGoing) OR #_w1;
   #State.Tank.ProWater.Ready_for_Inlet := #alwaysON AND #State.Tank.ProWater.Idle AND (#Parameter.SP_Prowater > 2.0) AND NOT #State.Tank.ProWater.OnGoing;
   IF #alwaysON AND #IN_FBAV_ProWater AND (#IN_FT_01 <= #Parameter.SP_Prowater) THEN
       #State.Tank.ProWater.OnGoing := TRUE;
   END_IF;
   IF #alwaysON AND #State.Tank.ProWater.OnGoing AND ((#IN_FBAV_ProWater AND (#IN_FT_01 > #Parameter.SP_Prowater)) OR NOT #IN_FBAV_ProWater) THEN
       #State.Tank.ProWater.OnGoing := FALSE;
   END_IF;
   #_w2 := #alwaysON AND NOT #State.Tank.ProWater.OnGoing AND #N_InletProOnGoing;   // falling edge of #State.Tank.ProWater.OnGoing
   #N_InletProOnGoing := #State.Tank.ProWater.OnGoing;
   IF #_w2 AND (#IN_FT_01 > #Parameter.SP_Prowater) THEN #State.Tank.ProWater.Done := TRUE; END_IF;
   IF #alwaysON AND #State.Tank.ProWater.OnGoing THEN #State.Tank.ProWater.Done := FALSE; END_IF;
END_REGION

REGION Network 3: Tank Status HotWater
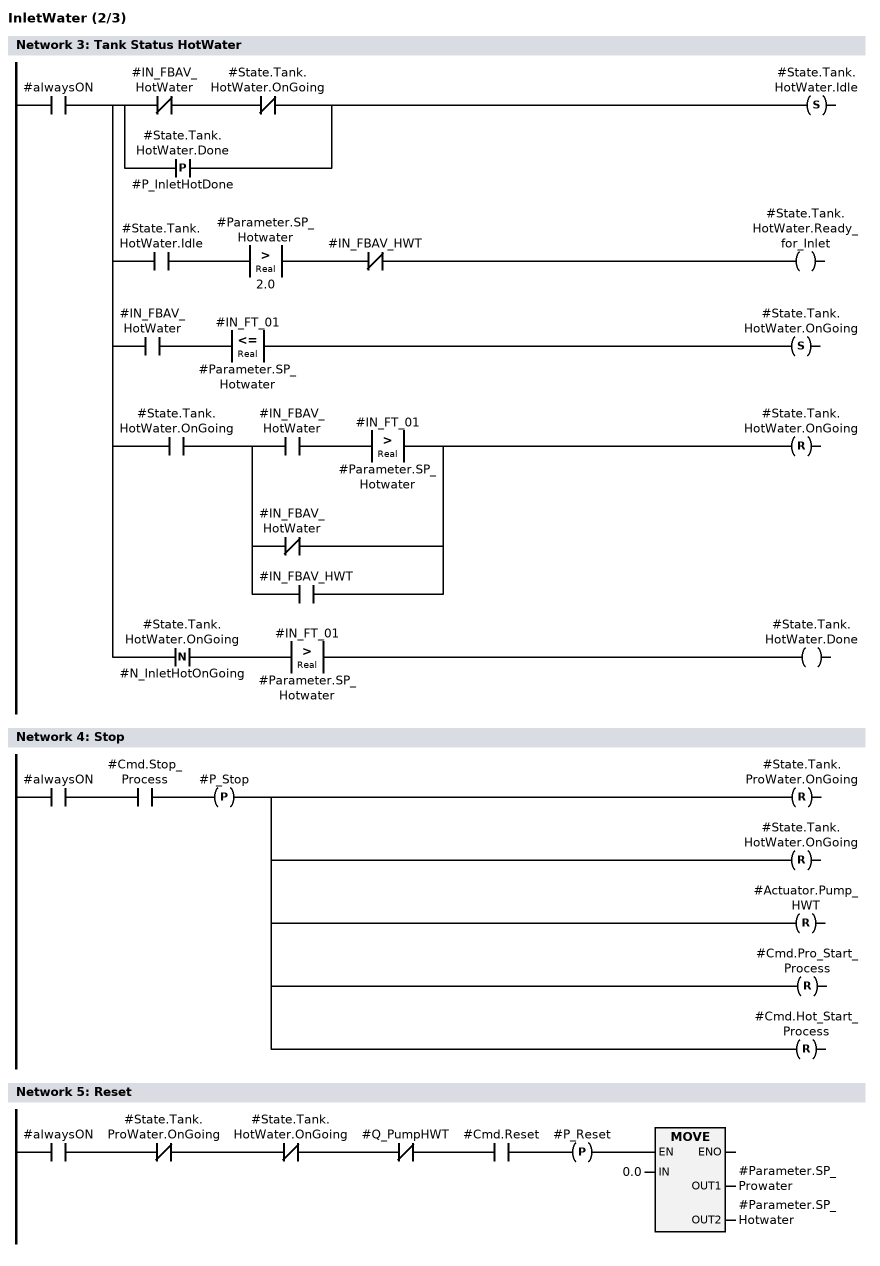
   RUNG wire#powerrail
      Contact( #alwaysON )
      wire#w1
      I_Contact( #IN_FBAV_HotWater )
      I_Contact( #State.Tank.HotWater.OnGoing )
      wire#w2
      S_Coil( #State.Tank.HotWater.Idle )
   END_RUNG
   RUNG wire#w1
      P_Contact(operand := #State.Tank.HotWater.Done, bit := #P_InletHotDone)
   END_RUNG wire#w2
   RUNG wire#w1
      Contact( #State.Tank.HotWater.Idle )
      { S7_Templates := "SrcType := Real" } GT_Contact(in1 := #Parameter.SP_Hotwater, in2 := 2.0)
      I_Contact( #IN_FBAV_HWT )
      Coil( #State.Tank.HotWater.Ready_for_Inlet )
   END_RUNG
   RUNG wire#w1
      Contact( #IN_FBAV_HotWater )
      { S7_Templates := "SrcType := Real" } LE_Contact(in1 := #IN_FT_01, in2 := #Parameter.SP_Hotwater)
      S_Coil( #State.Tank.HotWater.OnGoing )
   END_RUNG
   RUNG wire#w1
      Contact( #State.Tank.HotWater.OnGoing )
      wire#w3
      Contact( #IN_FBAV_HotWater )
      { S7_Templates := "SrcType := Real" } GT_Contact(in1 := #IN_FT_01, in2 := #Parameter.SP_Hotwater)
      wire#w4
      R_Coil( #State.Tank.HotWater.OnGoing )
   END_RUNG
   RUNG wire#w3
      I_Contact( #IN_FBAV_HotWater )
   END_RUNG wire#w4
   RUNG wire#w3
      Contact( #IN_FBAV_HWT )
   END_RUNG wire#w4
   RUNG wire#w1
      N_Contact(operand := #State.Tank.HotWater.OnGoing, bit := #N_InletHotOnGoing)
      { S7_Templates := "SrcType := Real" } GT_Contact(in1 := #IN_FT_01, in2 := #Parameter.SP_Hotwater)
      Coil( #State.Tank.HotWater.Done )
   END_RUNG
   // the same network as SCL:
   #_w1 := #alwaysON AND #State.Tank.HotWater.Done AND NOT #P_InletHotDone;   // rising edge of #State.Tank.HotWater.Done
   #P_InletHotDone := #State.Tank.HotWater.Done;
   IF (#alwaysON AND NOT #IN_FBAV_HotWater AND NOT #State.Tank.HotWater.OnGoing) OR #_w1 THEN
       #State.Tank.HotWater.Idle := TRUE;
   END_IF;
   #State.Tank.HotWater.Ready_for_Inlet := #alwaysON AND #State.Tank.HotWater.Idle AND (#Parameter.SP_Hotwater > 2.0) AND NOT #IN_FBAV_HWT;
   IF #alwaysON AND #IN_FBAV_HotWater AND (#IN_FT_01 <= #Parameter.SP_Hotwater) THEN
       #State.Tank.HotWater.OnGoing := TRUE;
   END_IF;
   IF #alwaysON AND #State.Tank.HotWater.OnGoing AND ((#IN_FBAV_HotWater AND (#IN_FT_01 > #Parameter.SP_Hotwater)) OR NOT #IN_FBAV_HotWater OR #IN_FBAV_HWT) THEN
       #State.Tank.HotWater.OnGoing := FALSE;
   END_IF;
   #_w2 := #alwaysON AND NOT #State.Tank.HotWater.OnGoing AND #N_InletHotOnGoing;   // falling edge of #State.Tank.HotWater.OnGoing
   #N_InletHotOnGoing := #State.Tank.HotWater.OnGoing;
   #State.Tank.HotWater.Done := #_w2 AND (#IN_FT_01 > #Parameter.SP_Hotwater);
END_REGION

REGION Network 4: Stop
   RUNG wire#powerrail
      Contact( #alwaysON )
      Contact( #Cmd.Stop_Process )
      P_Trig( #P_Stop )
      wire#w1
      R_Coil( #State.Tank.ProWater.OnGoing )
   END_RUNG
   RUNG wire#w1
      R_Coil( #State.Tank.HotWater.OnGoing )
   END_RUNG
   RUNG wire#w1
      R_Coil( #Actuator.Pump_HWT )
   END_RUNG
   RUNG wire#w1
      R_Coil( #Cmd.Pro_Start_Process )
   END_RUNG
   RUNG wire#w1
      R_Coil( #Cmd.Hot_Start_Process )
   END_RUNG
   // the same network as SCL:
   #_w1 := #alwaysON AND #Cmd.Stop_Process;
   #_w2 := #_w1 AND NOT #P_Stop;   // rising edge
   #P_Stop := #_w1;
   IF #_w2 THEN
       #State.Tank.ProWater.OnGoing := FALSE;
       #State.Tank.HotWater.OnGoing := FALSE;
       #Actuator.Pump_HWT := FALSE;
       #Cmd.Pro_Start_Process := FALSE;
       #Cmd.Hot_Start_Process := FALSE;
   END_IF;
END_REGION

REGION Network 5: Reset
   RUNG wire#powerrail
      Contact( #alwaysON )
      I_Contact( #State.Tank.ProWater.OnGoing )
      I_Contact( #State.Tank.HotWater.OnGoing )
      I_Contact( #Q_PumpHWT )
      Contact( #Cmd.Reset )
      P_Trig( #P_Reset )
      Move(in := 0.0, out1 => #Parameter.SP_Prowater, out2 => #Parameter.SP_Hotwater)
   END_RUNG
   // the same network as SCL:
   #_w1 := #alwaysON AND NOT #State.Tank.ProWater.OnGoing AND NOT #State.Tank.HotWater.OnGoing AND NOT #Q_PumpHWT AND #Cmd.Reset;
   #_w2 := #_w1 AND NOT #P_Reset;   // rising edge
   #P_Reset := #_w1;
   IF #_w2 THEN
       #Parameter.SP_Prowater := 0.0;
       #Parameter.SP_Hotwater := 0.0;
   END_IF;
END_REGION

REGION Network 6: Inlet ProWater
